C09088=1017.058,347.375,350.986,171.021,50.976,160.063
C09089=1017.051,347.128,351.023,171.013,50.980,160.063
C09090=1017.044,346.881,351.059,171.005,50.983,160.062
C09091=1017.036,346.634,351.096,170.997,50.986,160.061
C09092=1017.029,346.386,351.133,170.991,50.989,160.061
C09093=1017.022,346.139,351.168,170.983,50.992,160.060
C09094=1017.014,345.892,351.205,170.975,50.995,160.060
C09095=1017.007,345.644,351.241,170.967,50.998,160.059
C09096=1017.000,345.397,351.277,170.960,51.001,160.058
C09097=1016.992,345.150,351.314,170.953,51.004,160.058
C09098=1016.985,344.902,351.350,170.944,51.007,160.057
C09099=1016.978,344.655,351.386,170.938,51.010,160.057
C09100=1016.971,344.408,351.422,170.930,51.013,160.056
C09101=1016.964,344.161,351.458,170.922,51.017,160.056
C09102=1016.957,343.913,351.495,170.916,51.020,160.055
C09103=1016.949,343.666,351.531,170.908,51.023,160.054
C09104=1016.942,343.419,351.567,170.900,51.026,160.054
C09105=1016.935,343.171,351.604,170.892,51.029,160.053
C09106=1016.928,342.925,351.640,170.885,51.032,160.053
C09107=1016.921,342.677,351.675,170.878,51.036,160.052
C09108=1016.913,342.430,351.711,170.870,51.039,160.052
C09109=1016.907,342.182,351.748,170.863,51.042,160.051
C09110=1016.899,341.935,351.784,170.856,51.045,160.051
C09111=1016.892,341.687,351.819,170.848,51.049,160.050
C09112=1016.885,341.441,351.855,170.841,51.052,160.050
C09113=1016.878,341.193,351.892,170.833,51.055,160.049
C09114=1016.871,340.945,351.927,170.826,51.058,160.048
C09115=1016.864,340.699,351.963,170.819,51.061,160.048
C09116=1016.857,340.451,351.999,170.812,51.065,160.048
C09117=1016.850,340.204,352.034,170.804,51.069,160.047
C09118=1016.843,339.956,352.071,170.797,51.072,160.047
C09119=1016.836,339.709,352.106,170.790,51.075,160.046
C09120=1016.829,339.462,352.142,170.783,51.078,160.046
C09121=1016.822,339.214,352.178,170.775,51.081,160.045
C09122=1016.815,338.967,352.213,170.768,51.085,160.044
C09123=1016.808,338.720,352.249,170.761,51.088,160.044
C09124=1016.800,338.472,352.285,170.754,51.092,160.044
C09125=1016.793,338.225,352.320,170.746,51.096,160.043
C09126=1016.786,337.956,352.359,170.739,51.099,160.043
C09127=1016.778,337.686,352.397,170.731,51.103,160.042
C09128=1016.771,337.417,352.436,170.722,51.107,160.042
C09129=1016.763,337.148,352.474,170.715,51.111,160.041
C09130=1016.756,336.901,352.509,170.708,51.114,160.041
C09131=1016.749,336.653,352.545,170.701,51.117,160.040
C09132=1016.742,336.406,352.580,170.693,51.121,160.040
C09133=1016.735,336.158,352.615,170.687,51.125,160.040
C09134=1016.728,335.912,352.651,170.680,51.128,160.039
C09135=1016.721,335.664,352.686,170.672,51.132,160.039
C09136=1016.714,335.416,352.721,170.665,51.135,160.038
C09137=1016.707,335.169,352.757,170.658,51.139,160.038
C09138=1016.700,334.921,352.792,170.650,51.143,160.037
C09139=1016.694,334.674,352.827,170.644,51.146,160.037
C09140=1016.687,334.427,352.862,170.637,51.150,160.037
C09141=1016.680,334.179,352.897,170.630,51.153,160.036
C09142=1016.673,333.932,352.932,170.623,51.157,160.036
C09143=1016.667,333.685,352.967,170.616,51.161,160.035
C09144=1016.659,333.437,353.001,170.609,51.165,160.035
C09145=1016.652,333.189,353.037,170.601,51.168,160.035
C09146=1016.645,332.941,353.072,170.595,51.171,160.034
C09147=1016.639,332.694,353.107,170.588,51.176,160.034
C09148=1016.632,332.447,353.142,170.581,51.179,160.033
C09149=1016.625,332.199,353.177,170.574,51.183,160.033
C09150=1016.619,331.951,353.212,170.567,51.187,160.033
C09151=1016.611,331.704,353.246,170.560,51.190,160.032
C09152=1016.604,331.457,353.281,170.553,51.195,160.032
C09153=1016.598,331.209,353.316,170.547,51.198,160.032
C09154=1016.590,330.962,353.350,170.539,51.202,160.031
C09155=1016.584,330.714,353.385,170.532,51.206,160.031
C09156=1016.577,330.467,353.420,170.526,51.210,160.031
C09157=1016.570,330.220,353.453,170.518,51.214,160.031
C09158=1016.564,329.972,353.488,170.512,51.217,160.030
C09159=1016.557,329.724,353.523,170.505,51.221,160.030
C09160=1016.550,329.477,353.558,170.498,51.225,160.030
C09161=1016.543,329.229,353.592,170.491,51.229,160.029
C09162=1016.536,328.982,353.627,170.484,51.234,160.029
C09163=1016.530,328.734,353.661,170.477,51.237,160.029
C09164=1016.523,328.487,353.696,170.470,51.241,160.028
C09165=1016.517,328.240,353.730,170.464,51.245,160.028
C09166=1016.510,327.992,353.764,170.457,51.249,160.028
C09167=1016.503,327.744,353.799,170.451,51.253,160.028
C09168=1016.496,327.496,353.833,170.443,51.257,160.027
C09169=1016.490,327.248,353.868,170.437,51.261,160.027
C09170=1016.483,327.002,353.902,170.430,51.265,160.027
C09171=1016.476,326.754,353.936,170.423,51.269,160.026
C09172=1016.470,326.506,353.971,170.417,51.273,160.026
C09173=1016.463,326.258,354.005,170.409,51.277,160.026
C09174=1016.457,326.011,354.039,170.403,51.281,160.026
C09175=1016.450,325.764,354.072,170.396,51.285,160.025
C09176=1016.442,325.516,354.106,170.390,51.289,160.025
C09177=1016.437,325.269,354.140,170.383,51.293,160.025
C09178=1016.429,325.021,354.174,170.376,51.298,160.025
C09179=1016.422,324.773,354.208,170.370,51.302,160.024
C09180=1016.415,324.526,354.242,170.362,51.306,160.024
C09181=1016.408,324.279,354.275,170.357,51.311,160.024
C09182=1016.402,324.031,354.310,170.349,51.315,160.024
C09183=1016.395,323.783,354.343,170.342,51.319,160.024
C09184=1016.388,323.536,354.377,170.336,51.324,160.024
C09185=1016.381,323.288,354.410,170.329,51.328,160.023
C09186=1016.373,323.014,354.448,170.322,51.332,160.023
C09187=1016.367,322.741,354.485,170.314,51.337,160.023
C09188=1016.359,322.467,354.522,170.307,51.342,160.023
C09189=1016.352,322.194,354.559,170.300,51.346,160.022
C09190=1016.345,321.947,354.592,170.293,51.351,160.022
C09191=1016.339,321.699,354.627,170.286,51.355,160.022
C09192=1016.332,321.450,354.660,170.281,51.360,160.022
C09193=1016.325,321.203,354.693,170.273,51.364,160.022
C09194=1016.318,320.956,354.727,170.268,51.368,160.022
C09195=1016.312,320.708,354.760,170.260,51.373,160.021
C09196=1016.305,320.460,354.794,170.255,51.377,160.021
C09197=1016.298,320.213,354.828,170.247,51.381,160.021
C09198=1016.292,319.965,354.861,170.241,51.386,160.021
C09199=1016.285,319.718,354.894,170.235,51.391,160.021
C09200=1016.279,319.470,354.928,170.228,51.395,160.020
C09201=1016.272,319.222,354.961,170.222,51.399,160.020
C09202=1016.266,318.975,354.994,170.215,51.404,160.020
C09203=1016.259,318.727,355.028,170.209,51.408,160.020
C09204=1016.252,318.479,355.061,170.202,51.413,160.020
C09205=1016.246,318.231,355.094,170.196,51.417,160.020
C09206=1016.240,317.984,355.128,170.189,51.422,160.020
C09207=1016.233,317.736,355.161,170.183,51.426,160.020
C09208=1016.226,317.489,355.194,170.176,51.431,160.020
C09209=1016.221,317.241,355.228,170.170,51.435,160.019
C09210=1016.214,316.993,355.261,170.163,51.440,160.019
C09211=1016.207,316.745,355.294,170.157,51.445,160.019
C09212=1016.201,316.498,355.327,170.151,51.449,160.019
C09213=1016.195,316.250,355.360,170.144,51.453,160.019
C09214=1016.189,316.003,355.394,170.138,51.458,160.019
C09215=1016.182,315.755,355.427,170.131,51.463,160.019
C09216=1016.176,315.507,355.460,170.125,51.467,160.019
C09217=1016.169,315.259,355.492,170.119,51.472,160.019
C09218=1016.163,315.012,355.525,170.113,51.477,160.019
C09219=1016.156,314.764,355.560,170.106,51.481,160.018
C09220=1016.150,314.516,355.592,170.100,51.486,160.018
C09221=1016.144,314.269,355.625,170.093,51.491,160.018
C09222=1016.138,314.021,355.658,170.087,51.495,160.018
C09223=1016.131,313.774,355.691,170.080,51.500,160.018
C09224=1016.125,313.525,355.724,170.075,51.504,160.018
C09225=1016.119,313.277,355.757,170.068,51.509,160.018
C09226=1016.113,313.030,355.790,170.062,51.513,160.018
C09227=1016.106,312.783,355.823,170.055,51.518,160.018
C09228=1016.100,312.535,355.856,170.050,51.523,160.018
C09229=1016.094,312.287,355.889,170.043,51.528,160.018
C09230=1016.088,312.040,355.922,170.037,51.533,160.018
C09231=1016.082,311.792,355.955,170.031,51.538,160.018
C09232=1016.075,311.544,355.988,170.025,51.542,160.018
C09233=1016.069,311.297,356.020,170.018,51.547,160.018
C09234=1016.064,311.048,356.053,170.012,51.552,160.018
C09235=1016.057,310.801,356.086,170.005,51.557,160.017
C09236=1016.051,310.553,356.118,170.000,51.561,160.017
C09237=1016.045,310.306,356.151,169.993,51.566,160.017
C09238=1016.039,310.058,356.184,169.988,51.571,160.018
C09239=1016.032,309.810,356.217,169.981,51.576,160.017
C09240=1016.027,309.563,356.250,169.975,51.581,160.017
C09241=1016.021,309.314,356.282,169.968,51.585,160.017
C09242=1016.014,309.067,356.314,169.963,51.591,160.017
C09243=1016.008,308.819,356.346,169.956,51.595,160.017
C09244=1016.001,308.572,356.378,169.951,51.601,160.018
C09245=1015.995,308.323,356.410,169.944,51.606,160.017
C09246=1015.987,308.055,356.445,169.938,51.611,160.018
C09247=1015.980,307.787,356.480,169.931,51.617,160.018
C09248=1015.973,307.520,356.515,169.924,51.623,160.018
C09249=1015.966,307.252,356.550,169.917,51.628,160.018
C09250=1015.960,307.003,356.582,169.912,51.633,160.018
C09251=1015.953,306.756,356.613,169.905,51.638,160.018
C09252=1015.947,306.508,356.646,169.899,51.644,160.018
C09253=1015.940,306.260,356.677,169.893,51.648,160.018
C09254=1015.934,306.012,356.709,169.887,51.654,160.018
C09255=1015.928,305.765,356.740,169.882,51.659,160.018
C09256=1015.922,305.517,356.773,169.875,51.664,160.018
C09257=1015.915,305.269,356.805,169.868,51.669,160.018
C09258=1015.909,305.021,356.837,169.863,51.675,160.018
C09259=1015.903,304.773,356.869,169.856,51.680,160.018
C09260=1015.896,304.525,356.901,169.851,51.685,160.018
C09261=1015.890,304.277,356.933,169.845,51.690,160.019
C09262=1015.884,304.030,356.964,169.838,51.696,160.019
C09263=1015.878,303.782,356.996,169.832,51.700,160.019
C09264=1015.871,303.534,357.027,169.826,51.706,160.019
C09265=1015.865,303.286,357.059,169.821,51.711,160.019
C09266=1015.859,303.038,357.091,169.814,51.717,160.019
C09267=1015.853,302.790,357.122,169.808,51.722,160.019
C09268=1015.846,302.543,357.155,169.803,51.727,160.019
C09269=1015.840,302.295,357.187,169.796,51.733,160.019
C09270=1015.834,302.047,357.219,169.790,51.738,160.019
C09271=1015.828,301.799,357.250,169.784,51.743,160.019
C09272=1015.822,301.551,357.282,169.779,51.748,160.020
C09273=1015.815,301.303,357.313,169.772,51.754,160.020
C09274=1015.809,301.055,357.345,169.766,51.759,160.020
C09275=1015.803,300.808,357.376,169.761,51.765,160.020
C09276=1015.798,300.559,357.408,169.754,51.770,160.020
C09277=1015.791,300.311,357.439,169.749,51.775,160.020
C09278=1015.785,300.064,357.471,169.743,51.781,160.020
C09279=1015.779,299.816,357.502,169.737,51.786,160.021
C09280=1015.773,299.568,357.534,169.731,51.792,160.021
C09281=1015.767,299.320,357.565,169.725,51.797,160.021
C09282=1015.761,299.072,357.597,169.719,51.803,160.021
C09283=1015.755,298.825,357.629,169.713,51.808,160.021
C09284=1015.749,298.576,357.660,169.708,51.813,160.021
C09285=1015.743,298.328,357.691,169.702,51.820,160.022
C09286=1015.737,298.081,357.723,169.696,51.825,160.022
C09287=1015.731,297.832,357.755,169.690,51.830,160.022
C09288=1015.725,297.585,357.785,169.684,51.836,160.022
C09289=1015.719,297.336,357.817,169.678,51.841,160.022
C09290=1015.713,297.089,357.848,169.672,51.847,160.022
C09291=1015.707,296.841,357.880,169.667,51.853,160.023
C09292=1015.701,296.593,357.910,169.661,51.858,160.023
C09293=1015.695,296.345,357.943,169.655,51.864,160.023
C09294=1015.689,296.098,357.974,169.649,51.869,160.023
C09295=1015.683,295.849,358.005,169.643,51.875,160.023
C09296=1015.677,295.602,358.036,169.638,51.881,160.023
C09297=1015.671,295.353,358.067,169.631,51.886,160.024
C09298=1015.665,295.106,358.098,169.626,51.891,160.024
C09299=1015.659,294.857,358.130,169.620,51.898,160.024
C09300=1015.654,294.609,358.161,169.615,51.903,160.024
C09301=1015.648,294.362,358.192,169.608,51.908,160.024
C09302=1015.642,294.113,358.224,169.602,51.915,160.025
C09303=1015.636,293.866,358.255,169.597,51.920,160.025
C09304=1015.631,293.617,358.286,169.591,51.926,160.025
C09305=1015.624,293.370,358.317,169.586,51.931,160.025
C09306=1015.619,293.120,358.348,169.579,51.937,160.025
C09307=1015.613,292.869,358.380,169.575,51.943,160.026
C09308=1015.607,292.619,358.411,169.568,51.949,160.026
C09309=1015.601,292.370,358.442,169.562,51.955,160.026
C09310=1015.595,292.122,358.473,169.557,51.960,160.026
C09311=1015.589,291.873,358.503,169.551,51.966,160.027
C09312=1015.583,291.625,358.534,169.545,51.973,160.027
C09313=1015.578,291.378,358.565,169.540,51.978,160.027
C09314=1015.571,291.129,358.596,169.534,51.984,160.027
C09315=1015.565,290.882,358.626,169.528,51.990,160.028
C09316=1015.560,290.634,358.657,169.523,51.996,160.028
C09317=1015.553,290.385,358.688,169.517,52.002,160.028
C09318=1015.547,290.137,358.718,169.511,52.008,160.029
C09319=1015.541,289.890,358.748,169.505,52.013,160.029
C09320=1015.535,289.641,358.779,169.500,52.020,160.029
C09321=1015.529,289.393,358.809,169.494,52.026,160.029
C09322=1015.523,289.145,358.840,169.489,52.032,160.030
C09323=1015.517,288.897,358.870,169.483,52.038,160.030
C09324=1015.511,288.649,358.901,169.477,52.044,160.030
C09325=1015.505,288.401,358.931,169.472,52.050,160.030
C09326=1015.500,288.153,358.962,169.466,52.056,160.031
C09327=1015.494,287.905,358.993,169.460,52.062,160.031
C09328=1015.488,287.657,359.023,169.455,52.068,160.031
C09329=1015.482,287.409,359.053,169.449,52.074,160.032
C09330=1015.476,287.161,359.084,169.443,52.081,160.032
C09331=1015.471,286.913,359.113,169.438,52.087,160.032
C09332=1015.465,286.664,359.144,169.432,52.093,160.033
C09333=1015.459,286.416,359.174,169.426,52.099,160.033
C09334=1015.453,286.168,359.205,169.421,52.105,160.033
C09335=1015.446,285.921,359.235,169.416,52.112,160.034
C09336=1015.441,285.673,359.264,169.410,52.118,160.034
C09337=1015.435,285.425,359.295,169.404,52.124,160.034
C09338=1015.429,285.176,359.325,169.399,52.130,160.035
C09339=1015.423,284.928,359.355,169.393,52.136,160.035
C09340=1015.417,284.680,359.385,169.387,52.143,160.035
C09341=1015.411,284.432,359.416,169.382,52.149,160.036
C09342=1015.406,284.184,359.445,169.376,52.155,160.036
C09343=1015.400,283.936,359.476,169.371,52.162,160.037
C09344=1015.394,283.688,359.505,169.365,52.168,160.037
C09345=1015.388,283.440,359.535,169.360,52.174,160.037
C09346=1015.382,283.192,359.565,169.354,52.180,160.038
C09347=1015.377,282.944,359.595,169.349,52.187,160.038
C09348=1015.370,282.696,359.625,169.343,52.194,160.038
C09349=1015.364,282.447,359.655,169.338,52.200,160.039
C09350=1015.359,282.199,359.684,169.332,52.206,160.039
C09351=1015.353,281.951,359.715,169.327,52.213,160.040
C09352=1015.346,281.703,359.744,169.321,52.219,160.040
C09353=1015.341,281.455,359.774,169.316,52.225,160.040
C09354=1015.335,281.206,359.804,169.310,52.232,160.041
C09355=1015.329,280.958,359.833,169.304,52.238,160.041
C09356=1015.323,280.710,359.863,169.299,52.245,160.042
C09357=1015.318,280.462,359.893,169.294,52.251,160.042
C09358=1015.312,280.213,359.922,169.288,52.258,160.042
C09359=1015.305,279.966,359.952,169.283,52.265,160.043
C09360=1015.300,279.718,359.982,169.277,52.271,160.043
C09361=1015.294,279.469,360.011,169.271,52.278,160.044
C09362=1015.289,279.226,360.041,169.266,52.284,160.044
C09363=1015.283,278.984,360.069,169.261,52.290,160.044
C09364=1015.278,278.741,360.098,169.256,52.297,160.045
C09365=1015.272,278.498,360.127,169.250,52.303,160.045
C09366=1015.267,278.255,360.156,169.245,52.310,160.046
C09367=1015.261,278.012,360.185,169.240,52.316,160.046
C09368=1015.255,277.769,360.214,169.234,52.323,160.046
C09369=1015.249,277.526,360.243,169.230,52.329,160.047
C09370=1015.244,277.278,360.273,169.224,52.336,160.047
C09371=1015.239,277.030,360.302,169.218,52.343,160.048
C09372=1015.232,276.782,360.332,169.213,52.350,160.048
C09373=1015.227,276.534,360.361,169.208,52.355,160.049
C09374=1015.221,276.285,360.391,169.203,52.363,160.049
C09375=1015.215,276.037,360.420,169.197,52.370,160.050
C09376=1015.210,275.789,360.449,169.191,52.376,160.050
C09377=1015.204,275.541,360.478,169.186,52.383,160.050
C09378=1015.199,275.293,360.508,169.180,52.390,160.051
C09379=1015.192,275.045,360.537,169.176,52.397,160.052
C09380=1015.187,274.796,360.566,169.170,52.403,160.052
C09381=1015.181,274.548,360.595,169.165,52.410,160.052
C09382=1015.176,274.300,360.625,169.159,52.417,160.053
C09383=1015.170,274.052,360.653,169.154,52.424,160.053
C09384=1015.164,273.803,360.683,169.148,52.431,160.054
C09385=1015.158,273.555,360.712,169.143,52.438,160.054
C09386=1015.152,273.307,360.741,169.138,52.445,160.055
C09387=1015.147,273.059,360.770,169.133,52.451,160.055
C09388=1015.141,272.810,360.798,169.127,52.458,160.056
C09389=1015.135,272.562,360.828,169.122,52.465,160.056
C09390=1015.129,272.314,360.857,169.116,52.472,160.057
C09391=1015.124,272.066,360.886,169.111,52.479,160.057
C09392=1015.118,271.817,360.915,169.105,52.486,160.058
C09393=1015.113,271.569,360.944,169.101,52.493,160.059
C09394=1015.107,271.321,360.973,169.096,52.500,160.059
C09395=1015.101,271.073,361.001,169.090,52.507,160.060
C09396=1015.096,270.824,361.031,169.085,52.514,160.060
C09397=1015.090,270.577,361.060,169.079,52.521,160.061
C09398=1015.084,270.328,361.088,169.074,52.528,160.061
C09399=1015.078,270.080,361.118,169.068,52.535,160.062
C09400=1015.073,269.832,361.146,169.063,52.543,160.062
C09401=1015.068,269.583,361.175,169.058,52.550,160.063
C09402=1015.061,269.335,361.204,169.054,52.556,160.063
C09403=1015.056,269.087,361.232,169.048,52.564,160.064
C09404=1015.051,268.838,361.262,169.043,52.571,160.064
C09405=1015.045,268.590,361.290,169.037,52.578,160.065
C09406=1015.039,268.342,361.319,169.032,52.585,160.066
C09407=1015.033,268.094,361.347,169.027,52.592,160.066
C09408=1015.028,267.845,361.375,169.021,52.599,160.067
C09409=1015.022,267.597,361.405,169.016,52.607,160.067
C09410=1015.016,267.348,361.433,169.011,52.614,160.068
C09411=1015.011,267.100,361.461,169.006,52.621,160.068
C09412=1015.005,266.852,361.490,169.000,52.628,160.069
C09413=1015.000,266.604,361.519,168.995,52.636,160.070
C09414=1014.994,266.355,361.547,168.990,52.643,160.070
C09415=1014.988,266.108,361.576,168.984,52.650,160.071
C09416=1014.982,265.859,361.604,168.980,52.658,160.071
C09417=1014.977,265.611,361.632,168.974,52.665,160.072
C09418=1014.971,265.363,361.661,168.969,52.673,160.073
C09419=1014.966,265.114,361.689,168.964,52.680,160.073
C09420=1014.960,264.866,361.718,168.958,52.687,160.074
C09421=1014.955,264.617,361.746,168.953,52.695,160.074
C09422=1014.949,264.376,361.773,168.949,52.701,160.075
C09423=1014.943,264.136,361.801,168.944,52.709,160.076
C09424=1014.939,263.895,361.828,168.939,52.716,160.076
C09425=1014.933,263.654,361.855,168.933,52.723,160.077
C09426=1014.928,263.414,361.882,168.928,52.731,160.077
C09427=1014.922,263.174,361.910,168.924,52.738,160.078
C09428=1014.916,262.933,361.937,168.918,52.745,160.078
C09429=1014.911,262.692,361.965,168.914,52.753,160.079
C09430=1014.905,262.443,361.993,168.908,52.760,160.080
C09431=1014.900,262.195,362.021,168.903,52.767,160.080
C09432=1014.895,261.947,362.049,168.898,52.775,160.081
C09433=1014.889,261.698,362.077,168.893,52.782,160.082
C09434=1014.883,261.450,362.105,168.888,52.790,160.082
C09435=1014.877,261.202,362.134,168.883,52.798,160.083
C09436=1014.872,260.954,362.162,168.878,52.805,160.084
C09437=1014.867,260.705,362.190,168.873,52.813,160.084
C09438=1014.861,260.457,362.218,168.868,52.820,160.085
C09439=1014.855,260.209,362.246,168.863,52.828,160.086
C09440=1014.850,259.960,362.274,168.857,52.835,160.086
C09441=1014.844,259.711,362.301,168.852,52.843,160.087
C09442=1014.839,259.463,362.329,168.846,52.851,160.088
C09443=1014.834,259.215,362.357,168.841,52.859,160.088
C09444=1014.827,258.967,362.385,168.837,52.867,160.089
C09445=1014.822,258.719,362.413,168.832,52.875,160.090
C09446=1014.816,258.470,362.440,168.827,52.882,160.091
C09447=1014.810,258.222,362.468,168.822,52.890,160.091
C09448=1014.805,257.973,362.495,168.816,52.898,160.092
C09449=1014.799,257.725,362.523,168.811,52.906,160.093
C09450=1014.793,257.476,362.551,168.806,52.914,160.093
C09451=1014.787,257.228,362.578,168.801,52.922,160.094
C09452=1014.782,256.980,362.606,168.796,52.929,160.095
C09453=1014.776,256.731,362.633,168.790,52.938,160.095
C09454=1014.770,256.483,362.661,168.785,52.945,160.096
C09455=1014.765,256.234,362.688,168.780,52.953,160.097
C09456=1014.759,255.986,362.715,168.775,52.961,160.098
C09457=1014.753,255.737,362.743,168.770,52.969,160.098
C09458=1014.748,255.489,362.771,168.765,52.978,160.099
C09459=1014.742,255.241,362.797,168.760,52.985,160.100
C09460=1014.737,254.993,362.825,168.755,52.993,160.101
C09461=1014.731,254.743,362.853,168.750,53.001,160.101
C09462=1014.726,254.495,362.880,168.744,53.009,160.102
C09463=1014.720,254.247,362.908,168.740,53.018,160.103
C09464=1014.714,253.998,362.934,168.735,53.026,160.104
C09465=1014.709,253.750,362.962,168.730,53.033,160.104
C09466=1014.703,253.501,362.990,168.725,53.041,160.105
C09467=1014.698,253.253,363.016,168.719,53.049,160.106
C09468=1014.692,253.005,363.044,168.715,53.058,160.107
C09469=1014.687,252.756,363.071,168.710,53.066,160.107
C09470=1014.682,252.508,363.098,168.705,53.074,160.108
C09471=1014.676,252.260,363.126,168.700,53.082,160.109
C09472=1014.670,252.011,363.153,168.695,53.090,160.110
C09473=1014.665,251.762,363.181,168.690,53.098,160.110
C09474=1014.659,251.513,363.207,168.685,53.107,160.111
C09475=1014.654,251.265,363.235,168.679,53.115,160.112
C09476=1014.649,251.017,363.262,168.674,53.123,160.113
C09477=1014.643,250.768,363.289,168.670,53.131,160.114
C09478=1014.638,250.520,363.316,168.664,53.139,160.114
C09479=1014.632,250.272,363.344,168.660,53.148,160.115
C09480=1014.627,250.023,363.371,168.655,53.156,160.116
C09481=1014.622,249.775,363.398,168.650,53.164,160.117
C09482=1014.616,249.533,363.425,168.645,53.172,160.118
C09483=1014.611,249.291,363.451,168.641,53.180,160.118
C09484=1014.605,249.050,363.478,168.636,53.188,160.119
C09485=1014.600,248.808,363.504,168.630,53.196,160.120
C09486=1014.595,248.566,363.529,168.625,53.204,160.121
C09487=1014.590,248.325,363.556,168.620,53.212,160.121
C09488=1014.584,248.083,363.582,168.616,53.220,160.122
C09489=1014.579,247.841,363.609,168.611,53.229,160.123
C09490=1014.574,247.593,363.636,168.606,53.237,160.124
C09491=1014.568,247.344,363.663,168.602,53.245,160.125
C09492=1014.563,247.096,363.690,168.596,53.253,160.125
C09493=1014.558,246.847,363.717,168.592,53.262,160.126
C09494=1014.552,246.599,363.744,168.587,53.270,160.127
C09495=1014.547,246.350,363.771,168.581,53.279,160.128
C09496=1014.542,246.102,363.797,168.577,53.287,160.129
C09497=1014.537,245.854,363.825,168.572,53.295,160.129
C09498=1014.532,245.605,363.852,168.567,53.304,160.130
C09499=1014.526,245.357,363.879,168.562,53.312,160.131
C09500=1014.521,245.108,363.906,168.557,53.320,160.132
C09501=1014.515,244.860,363.932,168.552,53.329,160.133
C09502=1014.510,244.611,363.960,168.547,53.338,160.134
C09503=1014.505,244.362,363.987,168.543,53.346,160.134
C09504=1014.499,244.114,364.014,168.537,53.355,160.135
C09505=1014.494,243.865,364.041,168.533,53.363,160.136
C09506=1014.489,243.618,364.067,168.528,53.371,160.137
C09507=1014.484,243.368,364.094,168.522,53.380,160.138
C09508=1014.479,243.120,364.120,168.518,53.389,160.139
C09509=1014.474,242.871,364.148,168.514,53.397,160.140
C09510=1014.469,242.623,364.175,168.508,53.406,160.141
C09511=1014.463,242.374,364.201,168.503,53.414,160.141
C09512=1014.458,242.127,364.228,168.498,53.423,160.142
C09513=1014.452,241.878,364.254,168.494,53.432,160.143
C09514=1014.447,241.629,364.281,168.488,53.440,160.144
C09515=1014.441,241.381,364.308,168.484,53.449,160.145
C09516=1014.436,241.132,364.333,168.480,53.458,160.146
C09517=1014.431,240.884,364.360,168.474,53.467,160.147
C09518=1014.426,240.635,364.386,168.470,53.475,160.148
C09519=1014.420,240.386,364.413,168.464,53.484,160.148
C09520=1014.414,240.138,364.440,168.460,53.493,160.149
C09521=1014.410,239.889,364.466,168.455,53.502,160.150
C09522=1014.404,239.641,364.492,168.450,53.510,160.151
C09523=1014.399,239.392,364.518,168.445,53.519,160.152
C09524=1014.394,239.143,364.546,168.440,53.528,160.153
C09525=1014.388,238.894,364.572,168.436,53.538,160.154
C09526=1014.383,238.647,364.598,168.431,53.546,160.155
C09527=1014.378,238.398,364.624,168.426,53.555,160.156
C09528=1014.372,238.149,364.650,168.421,53.564,160.157
C09529=1014.367,237.901,364.676,168.416,53.573,160.158
C09530=1014.361,237.653,364.703,168.411,53.582,160.159
C09531=1014.356,237.404,364.729,168.407,53.591,160.160
C09532=1014.351,237.156,364.754,168.401,53.600,160.160
C09533=1014.345,236.907,364.781,168.397,53.609,160.161
C09534=1014.340,236.658,364.807,168.392,53.618,160.162
C09535=1014.334,236.409,364.833,168.387,53.627,160.163
C09536=1014.330,236.161,364.858,168.382,53.636,160.164
C09537=1014.324,235.913,364.885,168.378,53.646,160.165
C09538=1014.318,235.664,364.911,168.373,53.654,160.166
C09539=1014.313,235.415,364.936,168.368,53.663,160.167
C09540=1014.308,235.166,364.962,168.363,53.673,160.168
C09541=1014.302,234.918,364.989,168.359,53.681,160.169
C09542=1014.297,234.673,365.015,168.353,53.690,160.170
C09543=1014.293,234.428,365.040,168.349,53.700,160.171
C09544=1014.287,234.183,365.065,168.344,53.709,160.172
C09545=1014.282,233.938,365.091,168.340,53.717,160.173
C09546=1014.277,233.693,365.116,168.335,53.727,160.174
C09547=1014.271,233.448,365.141,168.329,53.736,160.175
C09548=1014.266,233.202,365.167,168.326,53.745,160.176
C09549=1014.261,232.957,365.193,168.320,53.754,160.177
C09550=1014.256,232.708,365.219,168.316,53.763,160.178
C09551=1014.251,232.460,365.244,168.311,53.773,160.179
C09552=1014.245,232.211,365.270,168.306,53.783,160.180
C09553=1014.240,231.963,365.295,168.302,53.791,160.181
C09554=1014.234,231.715,365.322,168.297,53.801,160.182
C09555=1014.229,231.466,365.347,168.292,53.810,160.183
C09556=1014.224,231.217,365.373,168.288,53.819,160.184
C09557=1014.219,230.969,365.399,168.283,53.828,160.185
C09558=1014.213,230.720,365.425,168.278,53.838,160.186
C09559=1014.208,230.472,365.450,168.273,53.848,160.187
C09560=1014.203,230.223,365.476,168.269,53.856,160.188
C09561=1014.198,229.974,365.501,168.264,53.866,160.189
C09562=1014.193,229.725,365.527,168.259,53.876,160.190
C09563=1014.188,229.477,365.553,168.255,53.885,160.191
C09564=1014.183,229.228,365.579,168.250,53.894,160.192
C09565=1014.177,228.980,365.603,168.245,53.904,160.193
C09566=1014.171,228.731,365.629,168.240,53.914,160.194
C09567=1014.167,228.482,365.655,168.235,53.923,160.195
C09568=1014.161,228.233,365.681,168.231,53.932,160.196
C09569=1014.157,227.984,365.706,168.226,53.942,160.197
C09570=1014.150,227.736,365.731,168.221,53.952,160.198
C09571=1014.146,227.488,365.757,168.216,53.961,160.199
C09572=1014.140,227.239,365.783,168.211,53.970,160.200
C09573=1014.135,226.990,365.807,168.207,53.980,160.202
C09574=1014.130,226.742,365.832,168.202,53.990,160.203
C09575=1014.124,226.493,365.858,168.198,53.999,160.204
C09576=1014.120,226.244,365.884,168.193,54.009,160.205
C09577=1014.114,225.995,365.909,168.188,54.019,160.206
C09578=1014.109,225.747,365.934,168.183,54.029,160.207
C09579=1014.104,225.499,365.960,168.178,54.038,160.208
C09580=1014.098,225.249,365.984,168.174,54.048,160.209
C09581=1014.093,225.001,366.010,168.170,54.058,160.210
C09582=1014.087,224.752,366.035,168.165,54.067,160.211
C09583=1014.082,224.503,366.060,168.160,54.077,160.212
C09584=1014.077,224.255,366.084,168.155,54.087,160.213
C09585=1014.072,224.006,366.110,168.151,54.097,160.215
C09586=1014.067,223.757,366.135,168.146,54.106,160.216
C09587=1014.061,223.509,366.160,168.141,54.117,160.217
C09588=1014.056,223.259,366.185,168.137,54.127,160.218
C09589=1014.051,223.011,366.210,168.132,54.137,160.219
C09590=1014.046,222.763,366.235,168.127,54.146,160.220
C09591=1014.040,222.513,366.260,168.122,54.156,160.221
C09592=1014.035,222.265,366.285,168.118,54.166,160.222
C09593=1014.030,222.016,366.310,168.113,54.176,160.223
C09594=1014.025,221.767,366.335,168.108,54.186,160.225
C09595=1014.019,221.519,366.360,168.104,54.196,160.226
C09596=1014.014,221.271,366.385,168.099,54.206,160.227
C09597=1014.009,221.021,366.410,168.094,54.216,160.228
C09598=1014.004,220.772,366.435,168.090,54.226,160.229
C09599=1013.998,220.524,366.460,168.085,54.236,160.230
C09600=1013.994,220.275,366.485,168.080,54.246,160.231
C09601=1013.988,220.026,366.509,168.076,54.256,160.232
C09602=1013.983,219.778,366.535,168.071,54.266,160.234
C09603=1013.978,219.529,366.559,168.067,54.276,160.235
C09604=1013.973,219.280,366.584,168.062,54.286,160.236
C09605=1013.969,219.032,366.609,168.057,54.296,160.237
C09606=1013.962,218.782,366.634,168.053,54.306,160.238
C09607=1013.957,218.532,366.659,168.048,54.316,160.239
C09608=1013.952,218.282,366.683,168.044,54.326,160.241
C09609=1013.947,218.032,366.709,168.039,54.336,160.242
C09610=1013.942,217.783,366.734,168.035,54.347,160.243
C09611=1013.937,217.535,366.758,168.030,54.357,160.244
C09612=1013.931,217.287,366.783,168.025,54.368,160.245
C09613=1013.926,217.038,366.807,168.020,54.377,160.246
C09614=1013.922,216.789,366.832,168.016,54.388,160.248
C09615=1013.916,216.540,366.856,168.011,54.398,160.249
C09616=1013.910,216.291,366.881,168.007,54.408,160.250
C09617=1013.905,216.043,366.905,168.002,54.418,160.251
C09618=1013.901,215.794,366.930,167.997,54.429,160.252
C09619=1013.895,215.545,366.954,167.992,54.440,160.254
C09620=1013.890,215.297,366.978,167.988,54.449,160.255
C09621=1013.885,215.048,367.003,167.984,54.460,160.256
C09622=1013.879,214.799,367.027,167.979,54.470,160.257
C09623=1013.874,214.550,367.052,167.975,54.480,160.259
C09624=1013.869,214.301,367.076,167.969,54.491,160.260
C09625=1013.864,214.053,367.101,167.965,54.501,160.261
C09626=1013.859,213.803,367.124,167.960,54.512,160.262
C09627=1013.854,213.555,367.149,167.956,54.522,160.263
C09628=1013.849,213.306,367.173,167.951,54.533,160.265
C09629=1013.843,213.057,367.198,167.946,54.543,160.266
C09630=1013.838,212.809,367.222,167.942,54.554,160.267
C09631=1013.833,212.560,367.246,167.938,54.564,160.268
C09632=1013.828,212.311,367.271,167.933,54.574,160.269
C09633=1013.823,212.063,367.295,167.928,54.585,160.271
C09634=1013.818,211.813,367.319,167.924,54.596,160.272
C09635=1013.813,211.565,367.343,167.920,54.606,160.273
C09636=1013.808,211.316,367.368,167.914,54.617,160.274
C09637=1013.803,211.067,367.392,167.910,54.627,160.276
C09638=1013.798,210.819,367.416,167.905,54.638,160.277
C09639=1013.792,210.570,367.441,167.901,54.648,160.278
C09640=1013.787,210.321,367.464,167.896,54.659,160.279
C09641=1013.783,210.072,367.489,167.892,54.670,160.281
C09642=1013.777,209.824,367.513,167.888,54.681,160.282
C09643=1013.772,209.575,367.537,167.883,54.691,160.283
C09644=1013.767,209.326,367.561,167.878,54.702,160.284
C09645=1013.762,209.077,367.585,167.874,54.712,160.286
C09646=1013.757,208.829,367.610,167.870,54.723,160.287
C09647=1013.752,208.579,367.633,167.864,54.734,160.288
C09648=1013.746,208.331,367.657,167.860,54.744,160.290
C09649=1013.741,208.082,367.681,167.855,54.755,160.291
C09650=1013.736,207.833,367.705,167.851,54.766,160.292
C09651=1013.731,207.584,367.729,167.847,54.777,160.293
C09652=1013.726,207.335,367.753,167.842,54.788,160.295
C09653=1013.720,207.087,367.777,167.837,54.798,160.296
C09654=1013.716,206.838,367.800,167.832,54.809,160.297
C09655=1013.711,206.590,367.825,167.829,54.821,160.299
C09656=1013.706,206.340,367.848,167.824,54.831,160.300
C09657=1013.700,206.092,367.872,167.819,54.842,160.301
C09658=1013.695,205.843,367.896,167.815,54.853,160.303
C09659=1013.690,205.594,367.920,167.810,54.864,160.304
C09660=1013.685,205.345,367.944,167.806,54.875,160.305
C09661=1013.681,205.096,367.967,167.801,54.886,160.306
C09662=1013.675,204.855,367.990,167.797,54.896,160.308
C09663=1013.670,204.612,368.014,167.792,54.907,160.309
C09664=1013.665,204.370,368.037,167.788,54.918,160.310
C09665=1013.661,204.128,368.060,167.783,54.929,160.312
C09666=1013.655,203.886,368.082,167.779,54.939,160.313
C09667=1013.650,203.644,368.105,167.775,54.950,160.314
C09668=1013.646,203.402,368.128,167.770,54.961,160.315
C09669=1013.640,203.160,368.151,167.766,54.972,160.317
C09670=1013.623,202.089,368.245,167.234,54.871,160.172
C09671=1013.619,201.841,368.267,167.229,54.883,160.173
C09672=1013.614,201.592,368.289,167.224,54.896,160.174
C09673=1013.611,201.342,368.311,167.219,54.908,160.176
C09674=1013.607,201.094,368.333,167.214,54.920,160.177
C09675=1013.603,200.844,368.354,167.210,54.932,160.179
C09676=1013.599,200.596,368.376,167.205,54.944,160.180
C09677=1013.595,200.347,368.399,167.201,54.956,160.182
C09678=1013.590,200.097,368.420,167.195,54.969,160.183
C09679=1013.587,199.849,368.442,167.191,54.980,160.184
C09680=1013.583,199.599,368.464,167.186,54.993,160.186
C09681=1013.579,199.351,368.485,167.182,55.005,160.187
C09682=1013.575,199.101,368.507,167.177,55.017,160.189
C09683=1013.571,198.852,368.529,167.173,55.029,160.190
C09684=1013.567,198.603,368.550,167.168,55.041,160.192
C09685=1013.562,198.355,368.572,167.162,55.053,160.193
C09686=1013.559,198.105,368.594,167.158,55.066,160.194
C09687=1013.555,197.856,368.614,167.153,55.078,160.196
C09688=1013.550,197.607,368.636,167.149,55.090,160.197
C09689=1013.546,197.359,368.657,167.144,55.102,160.199
C09690=1013.542,197.109,368.679,167.139,55.115,160.200
C09691=1013.538,196.860,368.700,167.135,55.127,160.201
C09692=1013.534,196.611,368.721,167.130,55.139,160.203
C09693=1013.530,196.363,368.742,167.126,55.151,160.204
C09694=1013.526,196.113,368.764,167.122,55.164,160.206
C09695=1013.521,195.863,368.785,167.117,55.176,160.207
C09696=1013.517,195.615,368.806,167.113,55.188,160.209
C09697=1013.514,195.365,368.828,167.107,55.200,160.210
C09698=1013.509,195.117,368.849,167.103,55.213,160.212
C09699=1013.505,194.867,368.870,167.098,55.225,160.213
C09700=1013.501,194.619,368.891,167.093,55.237,160.214
C09701=1013.497,194.369,368.913,167.089,55.249,160.216
C09702=1013.493,194.120,368.934,167.085,55.261,160.217
C09703=1013.489,193.871,368.954,167.081,55.274,160.219
C09704=1013.484,193.623,368.976,167.076,55.286,160.220
C09705=1013.481,193.374,368.998,167.072,55.298,160.222
C09706=1013.477,193.124,369.019,167.067,55.310,160.223
C09707=1013.473,192.875,369.040,167.062,55.322,160.225
C09708=1013.469,192.626,369.061,167.058,55.335,160.226
C09709=1013.465,192.377,369.082,167.054,55.347,160.228
C09710=1013.461,192.128,369.103,167.050,55.359,160.229
C09711=1013.457,191.879,369.124,167.045,55.371,160.231
C09712=1013.454,191.630,369.145,167.040,55.383,160.232
C09713=1013.449,191.380,369.167,167.036,55.396,160.234
C09714=1013.445,191.132,369.187,167.032,55.407,160.235
C09715=1013.441,190.882,369.208,167.027,55.419,160.236
C09716=1013.437,190.633,369.230,167.023,55.432,160.238
C09717=1013.433,190.384,369.251,167.018,55.444,160.239
C09718=1013.429,190.135,369.272,167.014,55.456,160.241
C09719=1013.426,189.886,369.293,167.010,55.468,160.242
C09720=1013.422,189.637,369.314,167.005,55.480,160.244
C09721=1013.417,189.388,369.335,167.001,55.493,160.245
C09722=1013.413,189.139,369.356,166.996,55.505,160.247
C09723=1013.410,188.890,369.377,166.992,55.517,160.248
C09724=1013.406,188.641,369.398,166.988,55.529,160.250
C09725=1013.402,188.392,369.419,166.983,55.541,160.251
C09726=1013.398,188.143,369.440,166.979,55.553,160.252
C09727=1013.394,187.893,369.462,166.975,55.566,160.254
C09728=1013.390,187.645,369.482,166.970,55.578,160.255
C09729=1013.386,187.396,369.503,166.966,55.590,160.257
C09730=1013.382,187.146,369.524,166.962,55.601,160.258
C09731=1013.378,186.868,369.548,166.957,55.615,160.260
C09732=1013.374,186.589,369.571,166.953,55.629,160.262
C09733=1013.369,186.309,369.595,166.948,55.642,160.263
C09734=1013.365,186.030,369.618,166.943,55.656,160.265
C09735=1013.361,185.781,369.638,166.939,55.668,160.266
C09736=1013.357,185.532,369.659,166.935,55.681,160.268
C09737=1013.354,185.283,369.681,166.930,55.693,160.269
C09738=1013.350,185.034,369.702,166.926,55.704,160.271
C09739=1013.346,184.785,369.723,166.922,55.716,160.272
C09740=1013.342,184.536,369.743,166.918,55.729,160.274
C09741=1013.339,184.286,369.764,166.913,55.741,160.275
C09742=1013.335,184.038,369.785,166.909,55.753,160.277
C09743=1013.331,183.788,369.806,166.905,55.764,160.278
C09744=1013.327,183.540,369.827,166.901,55.776,160.279
C09745=1013.324,183.290,369.847,166.897,55.789,160.281
C09746=1013.320,183.041,369.868,166.892,55.801,160.282
C09747=1013.316,182.792,369.889,166.889,55.813,160.284
C09748=1013.313,182.543,369.910,166.884,55.825,160.285
C09749=1013.309,182.293,369.931,166.880,55.837,160.287
C09750=1013.305,182.045,369.952,166.877,55.849,160.289
C09751=1013.301,181.795,369.972,166.873,55.861,160.290
C09752=1013.298,181.546,369.993,166.868,55.873,160.291
C09753=1013.293,181.297,370.014,166.864,55.885,160.293
C09754=1013.289,181.048,370.034,166.860,55.898,160.294
C09755=1013.285,180.798,370.054,166.856,55.909,160.296
C09756=1013.282,180.549,370.074,166.852,55.922,160.297
C09757=1013.277,180.301,370.094,166.848,55.934,160.299
C09758=1013.274,180.051,370.114,166.844,55.947,160.300
C09759=1013.269,179.801,370.134,166.839,55.959,160.302
C09760=1013.265,179.553,370.155,166.835,55.971,160.303
C09761=1013.261,179.303,370.175,166.831,55.983,160.305
C09762=1013.257,179.054,370.194,166.828,55.995,160.306
C09763=1013.253,178.805,370.214,166.824,56.008,160.308
C09764=1013.249,178.557,370.234,166.819,56.020,160.309
C09765=1013.245,178.307,370.254,166.815,56.032,160.311
C09766=1013.241,178.058,370.275,166.811,56.045,160.312
C09767=1013.236,177.808,370.294,166.807,56.056,160.314
C09768=1013.233,177.559,370.314,166.804,56.069,160.316
C09769=1013.228,177.310,370.335,166.799,56.081,160.317
C09770=1013.224,177.061,370.355,166.795,56.093,160.318
C09771=1013.220,176.812,370.374,166.792,56.105,160.320
C09772=1013.217,176.563,370.394,166.787,56.118,160.322
C09773=1013.213,176.313,370.414,166.783,56.130,160.323
C09774=1013.208,176.065,370.434,166.779,56.142,160.325
C09775=1013.205,175.815,370.455,166.776,56.154,160.326
C09776=1013.200,175.566,370.474,166.771,56.166,160.328
C09777=1013.197,175.317,370.494,166.767,56.179,160.329
C09778=1013.193,175.068,370.514,166.764,56.191,160.331
C09779=1013.189,174.819,370.534,166.760,56.203,160.332
C09780=1013.185,174.569,370.554,166.756,56.215,160.334
C09781=1013.181,174.320,370.573,166.752,56.227,160.335
C09782=1013.177,174.071,370.593,166.748,56.239,160.337
C09783=1013.173,173.822,370.614,166.744,56.251,160.338
C09784=1013.169,173.573,370.633,166.741,56.264,160.340
C09785=1013.165,173.324,370.654,166.736,56.276,160.341
C09786=1013.161,173.075,370.673,166.732,56.288,160.343
C09787=1013.157,172.825,370.693,166.729,56.299,160.344
C09788=1013.154,172.576,370.713,166.725,56.312,160.346
C09789=1013.149,172.327,370.733,166.722,56.324,160.347
C09790=1013.146,172.078,370.753,166.717,56.336,160.349
C09791=1013.141,171.829,370.772,166.713,56.348,160.350
C09792=1013.138,171.579,370.792,166.710,56.361,160.352
C09793=1013.133,171.330,370.812,166.706,56.373,160.353
C09794=1013.130,171.081,370.832,166.702,56.384,160.355
C09795=1013.126,170.802,370.854,166.698,56.398,160.357
C09796=1013.121,170.522,370.876,166.693,56.412,160.358
C09797=1013.117,170.244,370.898,166.690,56.425,160.360
C09798=1013.113,169.965,370.920,166.685,56.438,160.362
C09799=1013.109,169.715,370.940,166.681,56.451,160.363
C09800=1013.105,169.466,370.960,166.678,56.462,160.365
C09801=1013.101,169.217,370.979,166.674,56.475,160.366
C09802=1013.097,168.968,371.000,166.671,56.487,160.368
C09803=1013.093,168.719,371.019,166.666,56.499,160.369
C09804=1013.089,168.469,371.039,166.663,56.511,160.371
C09805=1013.086,168.220,371.059,166.660,56.522,160.372
C09806=1013.082,167.971,371.078,166.655,56.535,160.374
C09807=1013.079,167.722,371.098,166.652,56.546,160.375
C09808=1013.074,167.473,371.117,166.648,56.558,160.377
C09809=1013.071,167.223,371.137,166.645,56.570,160.378
C09810=1013.066,166.974,371.157,166.640,56.582,160.380
C09811=1013.063,166.725,371.177,166.638,56.595,160.382
C09812=1013.060,166.476,371.196,166.634,56.607,160.383
C09813=1013.056,166.227,371.215,166.630,56.619,160.385
C09814=1013.052,165.977,371.235,166.627,56.630,160.386
C09815=1013.048,165.728,371.255,166.623,56.643,160.388
C09816=1013.044,165.479,371.275,166.619,56.654,160.389
C09817=1013.041,165.229,371.295,166.616,56.666,160.391
C09818=1013.037,164.981,371.314,166.612,56.678,160.392
C09819=1013.034,164.731,371.333,166.609,56.690,160.394
C09820=1013.029,164.482,371.353,166.605,56.702,160.395
C09821=1013.026,164.233,371.373,166.601,56.714,160.397
C09822=1013.022,163.984,371.392,166.598,56.726,160.398
C09823=1013.019,163.734,371.411,166.595,56.737,160.400
C09824=1013.015,163.485,371.431,166.590,56.750,160.401
C09825=1013.011,163.236,371.451,166.587,56.761,160.403
C09826=1013.007,162.987,371.471,166.584,56.773,160.404
C09827=1013.004,162.738,371.489,166.581,56.785,160.406
C09828=1013.000,162.488,371.509,166.576,56.796,160.407
C09829=1012.996,162.239,371.529,166.573,56.808,160.409
C09830=1012.993,161.991,371.548,166.570,56.820,160.410
C09831=1012.989,161.741,371.568,166.566,56.832,160.412
C09832=1012.985,161.492,371.587,166.562,56.844,160.413
C09833=1012.981,161.242,371.607,166.559,56.856,160.415
C09834=1012.978,160.993,371.626,166.556,56.867,160.416
C09835=1012.974,160.744,371.646,166.553,56.879,160.418
C09836=1012.971,160.495,371.666,166.550,56.891,160.420
C09837=1012.967,160.246,371.684,166.545,56.903,160.421
C09838=1012.964,159.996,371.704,166.542,56.914,160.422
C09839=1012.959,159.747,371.724,166.539,56.926,160.424
C09840=1012.956,159.497,371.743,166.535,56.938,160.425
C09841=1012.952,159.249,371.762,166.532,56.950,160.427
C09842=1012.949,159.000,371.782,166.529,56.962,160.429
C09843=1012.945,158.750,371.802,166.525,56.973,160.430
C09844=1012.942,158.501,371.821,166.521,56.985,160.431
C09845=1012.938,158.251,371.840,166.518,56.997,160.433
C09846=1012.934,158.002,371.860,166.515,57.008,160.435
C09847=1012.930,157.753,371.878,166.512,57.020,160.436
C09848=1012.926,157.504,371.897,166.509,57.032,160.438
C09849=1012.923,157.254,371.917,166.505,57.044,160.439
C09850=1012.919,157.005,371.936,166.501,57.056,160.441
C09851=1012.915,156.756,371.954,166.498,57.068,160.442
C09852=1012.911,156.507,371.973,166.495,57.079,160.444
C09853=1012.908,156.258,371.992,166.491,57.091,160.445
C09854=1012.903,156.008,372.011,166.487,57.103,160.447
C09855=1012.899,155.759,372.030,166.484,57.115,160.448
C09856=1012.896,155.510,372.048,166.481,57.127,160.450
C09857=1012.892,155.260,372.067,166.478,57.139,160.451
C09858=1012.888,155.011,372.086,166.475,57.151,160.453
C09859=1012.883,154.732,372.108,166.471,57.164,160.455
C09860=1012.880,154.452,372.129,166.467,57.177,160.456
C09861=1012.875,154.173,372.150,166.463,57.190,160.458
C09862=1012.871,153.894,372.171,166.460,57.203,160.460
C09863=1012.868,153.645,372.189,166.457,57.215,160.461
C09864=1012.863,153.396,372.209,166.454,57.227,160.463
C09865=1012.859,153.146,372.228,166.451,57.239,160.465
C09866=1012.856,152.897,372.246,166.447,57.250,160.466
C09867=1012.852,152.647,372.265,166.443,57.262,160.467
C09868=1012.848,152.399,372.283,166.440,57.274,160.469
C09869=1012.844,152.149,372.302,166.437,57.286,160.471
C09870=1012.840,151.899,372.321,166.434,57.298,160.472
C09871=1012.837,151.651,372.340,166.431,57.309,160.474
C09872=1012.832,151.401,372.358,166.427,57.321,160.475
C09873=1012.829,151.152,372.377,166.424,57.332,160.477
C09874=1012.825,150.903,372.396,166.421,57.344,160.478
C09875=1012.822,150.654,372.414,166.418,57.356,160.480
C09876=1012.818,150.404,372.433,166.415,57.368,160.482
C09877=1012.814,150.155,372.451,166.411,57.379,160.483
C09878=1012.810,149.905,372.470,166.408,57.391,160.484
C09879=1012.807,149.656,372.488,166.405,57.403,160.486
C09880=1012.803,149.407,372.507,166.402,57.414,160.487
C09881=1012.799,149.158,372.525,166.399,57.426,160.489
C09882=1012.795,148.908,372.544,166.396,57.438,160.491
C09883=1012.791,148.659,372.562,166.393,57.450,160.492
C09884=1012.787,148.410,372.581,166.389,57.461,160.494
C09885=1012.783,148.161,372.599,166.386,57.473,160.495
C09886=1012.779,147.911,372.618,166.383,57.485,160.497
C09887=1012.776,147.662,372.636,166.380,57.496,160.498
C09888=1012.772,147.413,372.655,166.377,57.508,160.500
C09889=1012.768,147.164,372.673,166.373,57.519,160.501
C09890=1012.764,146.914,372.692,166.370,57.531,160.503
C09891=1012.761,146.665,372.711,166.368,57.542,160.505
C09892=1012.757,146.415,372.729,166.365,57.554,160.506
C09893=1012.753,146.167,372.747,166.362,57.565,160.508
C09894=1012.749,145.916,372.765,166.359,57.577,160.509
C09895=1012.746,145.667,372.784,166.355,57.589,160.511
C09896=1012.742,145.418,372.802,166.352,57.601,160.512
C09897=1012.738,145.169,372.821,166.349,57.612,160.513
C09898=1012.734,144.919,372.839,166.346,57.624,160.515
C09899=1012.730,144.670,372.857,166.344,57.635,160.517
C09900=1012.727,144.421,372.875,166.340,57.646,160.518
C09901=1012.723,144.171,372.894,166.337,57.658,160.520
C09902=1012.718,143.923,372.911,166.334,57.669,160.521
C09903=1012.714,143.673,372.930,166.331,57.681,160.523
C09904=1012.711,143.423,372.948,166.328,57.693,160.525
C09905=1012.707,143.175,372.966,166.324,57.705,160.526
C09906=1012.703,142.925,372.984,166.321,57.716,160.528
C09907=1012.700,142.675,373.002,166.319,57.727,160.529
C09908=1012.695,142.426,373.020,166.316,57.739,160.531
C09909=1012.692,142.177,373.039,166.313,57.750,160.532
C09910=1012.688,141.928,373.056,166.310,57.762,160.534
C09911=1012.684,141.678,373.074,166.306,57.774,160.535
C09912=1012.680,141.429,373.093,166.304,57.785,160.537
C09913=1012.676,141.179,373.110,166.301,57.796,160.538
C09914=1012.672,140.930,373.129,166.298,57.808,160.540
C09915=1012.669,140.681,373.147,166.294,57.820,160.541
C09916=1012.665,140.431,373.165,166.293,57.831,160.543
C09917=1012.661,140.182,373.183,166.289,57.842,160.544
C09918=1012.658,139.933,373.201,166.286,57.854,160.546
C09919=1012.653,139.683,373.219,166.284,57.865,160.548
C09920=1012.650,139.434,373.237,166.280,57.876,160.549
C09921=1012.646,139.186,373.256,166.278,57.888,160.551
C09922=1012.642,138.936,373.273,166.275,57.899,160.552
C09923=1012.638,138.638,373.295,166.271,57.913,160.554
C09924=1012.633,138.340,373.316,166.268,57.927,160.556
C09925=1012.628,138.042,373.338,166.265,57.940,160.558
C09926=1012.624,137.745,373.359,166.260,57.953,160.559
C09927=1012.621,137.495,373.377,166.259,57.965,160.561
C09928=1012.617,137.245,373.396,166.255,57.976,160.562
C09929=1012.613,136.996,373.413,166.252,57.987,160.564
C09930=1012.609,136.747,373.431,166.250,57.999,160.566
C09931=1012.605,136.497,373.449,166.247,58.010,160.567
C09932=1012.602,136.248,373.466,166.244,58.021,160.568
C09933=1012.598,135.999,373.484,166.241,58.033,160.570
C09934=1012.593,135.749,373.502,166.238,58.044,160.572
C09935=1012.590,135.500,373.520,166.236,58.055,160.573
C09936=1012.586,135.251,373.537,166.232,58.066,160.574
C09937=1012.582,135.002,373.555,166.230,58.078,160.576
C09938=1012.578,134.752,373.573,166.227,58.089,160.578
C09939=1012.546,148.398,372.188,166.347,57.641,160.519
C09940=1012.549,148.647,372.170,166.351,57.630,160.518
C09941=1012.553,148.897,372.151,166.353,57.619,160.516
C09942=1012.557,149.145,372.133,166.356,57.607,160.514
C09943=1012.561,149.395,372.114,166.359,57.596,160.513
C09944=1012.564,149.644,372.096,166.362,57.584,160.511
C09945=1012.569,149.893,372.077,166.366,57.572,160.510
C09946=1012.572,150.142,372.059,166.369,57.561,160.509
C09947=1012.576,150.392,372.040,166.372,57.549,160.507
C09948=1012.580,150.641,372.022,166.375,57.537,160.506
C09949=1012.584,150.891,372.003,166.378,57.526,160.504
C09950=1012.587,151.140,371.985,166.381,57.514,160.502
C09951=1012.591,151.389,371.966,166.385,57.502,160.501
C09952=1012.595,151.638,371.948,166.388,57.491,160.499
C09953=1012.598,151.887,371.929,166.391,57.479,160.498
C09954=1012.602,152.137,371.910,166.394,57.467,160.496
C09955=1012.606,152.386,371.892,166.397,57.456,160.495
C09956=1012.610,152.636,371.873,166.400,57.444,160.493
C09957=1012.613,152.884,371.855,166.404,57.433,160.492
C09958=1012.617,153.134,371.836,166.407,57.421,160.490
C09959=1012.621,153.384,371.817,166.410,57.409,160.489
C09960=1012.627,153.781,371.787,166.416,57.390,160.486
C09961=1012.633,154.179,371.758,166.421,57.372,160.484
C09962=1012.638,154.577,371.727,166.426,57.353,160.481
C09963=1012.644,154.976,371.697,166.431,57.334,160.479
C09964=1012.648,155.226,371.679,166.434,57.322,160.477
C09965=1012.652,155.474,371.659,166.437,57.311,160.476
C09966=1012.656,155.724,371.641,166.440,57.299,160.474
C09967=1012.660,155.972,371.622,166.445,57.287,160.473
C09968=1012.664,156.222,371.604,166.448,57.275,160.471
C09969=1012.667,156.471,371.585,166.451,57.263,160.470
C09970=1012.671,156.720,371.566,166.454,57.252,160.468
C09971=1012.676,156.970,371.547,166.457,57.240,160.467
C09972=1012.678,157.219,371.528,166.460,57.228,160.465
C09973=1012.682,157.469,371.509,166.465,57.216,160.464
C09974=1012.686,157.717,371.490,166.468,57.204,160.462
C09975=1012.690,157.967,371.471,166.471,57.193,160.461
C09976=1012.694,158.216,371.453,166.474,57.181,160.459
C09977=1012.697,158.465,371.433,166.477,57.169,160.457
C09978=1012.700,158.715,371.414,166.481,57.158,160.456
C09979=1012.705,158.964,371.394,166.485,57.145,160.455
C09980=1012.707,159.213,371.375,166.488,57.134,160.453
C09981=1012.712,159.462,371.356,166.491,57.122,160.451
C09982=1012.715,159.712,371.336,166.495,57.111,160.450
C09983=1012.719,159.961,371.317,166.498,57.099,160.449
C09984=1012.722,160.211,371.298,166.501,57.087,160.447
C09985=1012.726,160.460,371.278,166.504,57.075,160.445
C09986=1012.730,160.708,371.259,166.507,57.063,160.444
C09987=1012.733,160.958,371.239,166.512,57.052,160.443
C09988=1012.737,161.207,371.220,166.515,57.040,160.441
C09989=1012.740,161.457,371.201,166.518,57.028,160.439
C09990=1012.744,161.706,371.181,166.521,57.016,160.438
C09991=1012.747,161.954,371.162,166.524,57.005,160.436
C09992=1012.751,162.204,371.142,166.529,56.993,160.435
C09993=1012.755,162.453,371.123,166.532,56.981,160.434
C09994=1012.758,162.703,371.103,166.535,56.969,160.432
C09995=1012.762,162.952,371.084,166.539,56.958,160.430
C09996=1012.766,163.201,371.064,166.543,56.945,160.429
//INST
///DATE 2021/06/25 14:50
///ATTR SC,RW,RJ
////FRAME ROBOT
///GROUP1 RB1
NOP
MOVL C00000 V=800.0 PL=0
MOVL C00001 V=800.0 PL=0
MOVL C00002 V=800.0 PL=0
MOVL C00003 V=800.0 PL=0
MOVL C00004 V=800.0 PL=0
MOVL C00005 V=800.0 PL=0
MOVL C00006 V=800.0 PL=0
MOVL C00007 V=800.0 PL=0
MOVL C00008 V=800.0 PL=0
MOVL C00009 V=800.0 PL=0
MOVL C00010 V=800.0 PL=0
MOVL C00011 V=800.0 PL=0
MOVL C00012 V=800.0 PL=0
MOVL C00013 V=800.0 PL=0
MOVL C00014 V=800.0 PL=0
MOVL C00015 V=800.0 PL=0
MOVL C00016 V=800.0 PL=0
MOVL C00017 V=800.0 PL=0
MOVL C00018 V=800.0 PL=0
MOVL C00019 V=800.0 PL=0
MOVL C00020 V=800.0 PL=0
MOVL C00021 V=800.0 PL=0
MOVL C00022 V=800.0 PL=0
MOVL C00023 V=800.0 PL=0
MOVL C00024 V=800.0 PL=0
MOVL C00025 V=800.0 PL=0
MOVL C00026 V=800.0 PL=0
MOVL C00027 V=800.0 PL=0
MOVL C00028 V=800.0 PL=0
MOVL C00029 V=800.0 PL=0
MOVL C00030 V=800.0 PL=0
MOVL C00031 V=800.0 PL=0
MOVL C00032 V=800.0 PL=0
MOVL C00033 V=800.0 PL=0
MOVL C00034 V=800.0 PL=0
MOVL C00035 V=800.0 PL=0
MOVL C00036 V=800.0 PL=0
MOVL C00037 V=800.0 PL=0
MOVL C00038 V=800.0 PL=0
MOVL C00039 V=800.0 PL=0
MOVL C00040 V=800.0 PL=0
MOVL C00041 V=800.0 PL=0
MOVL C00042 V=800.0 PL=0
MOVL C00043 V=800.0 PL=0
MOVL C00044 V=800.0 PL=0
MOVL C00045 V=800.0 PL=0
MOVL C00046 V=800.0 PL=0
MOVL C00047 V=800.0 PL=0
MOVL C00048 V=800.0 PL=0
MOVL C00049 V=800.0 PL=0
MOVL C00050 V=800.0 PL=0
MOVL C00051 V=800.0 PL=0
MOVL C00052 V=800.0 PL=0
MOVL C00053 V=800.0 PL=0
MOVL C00054 V=800.0 PL=0
MOVL C00055 V=800.0 PL=0
MOVL C00056 V=800.0 PL=0
MOVL C00057 V=800.0 PL=0
MOVL C00058 V=800.0 PL=0
MOVL C00059 V=800.0 PL=0
MOVL C00060 V=800.0 PL=0
MOVL C00061 V=800.0 PL=0
MOVL C00062 V=800.0 PL=0
MOVL C00063 V=800.0 PL=0
MOVL C00064 V=800.0 PL=0
MOVL C00065 V=800.0 PL=0
MOVL C00066 V=800.0 PL=0
MOVL C00067 V=800.0 PL=0
MOVL C00068 V=800.0 PL=0
MOVL C00069 V=800.0 PL=0
MOVL C00070 V=800.0 PL=0
MOVL C00071 V=800.0 PL=0
MOVL C00072 V=800.0 PL=0
MOVL C00073 V=800.0 PL=0
MOVL C00074 V=800.0 PL=0
MOVL C00075 V=800.0 PL=0
MOVL C00076 V=800.0 PL=0
MOVL C00077 V=800.0 PL=0
MOVL C00078 V=800.0 PL=0
MOVL C00079 V=800.0 PL=0
MOVL C00080 V=800.0 PL=0
MOVL C00081 V=800.0 PL=0
MOVL C00082 V=800.0 PL=0
MOVL C00083 V=800.0 PL=0
MOVL C00084 V=800.0 PL=0
MOVL C00085 V=800.0 PL=0
MOVL C00086 V=800.0 PL=0
MOVL C00087 V=800.0 PL=0
MOVL C00088 V=800.0 PL=0
MOVL C00089 V=800.0 PL=0
MOVL C00090 V=800.0 PL=0
MOVL C00091 V=800.0 PL=0
MOVL C00092 V=800.0 PL=0
MOVL C00093 V=800.0 PL=0
MOVL C00094 V=800.0 PL=0
MOVL C00095 V=800.0 PL=0
MOVL C00096 V=800.0 PL=0
MOVL C00097 V=800.0 PL=0
MOVL C00098 V=800.0 PL=0
MOVL C00099 V=800.0 PL=0
MOVL C00100 V=800.0 PL=0
MOVL C00101 V=800.0 PL=0
MOVL C00102 V=800.0 PL=0
MOVL C00103 V=800.0 PL=0
MOVL C00104 V=800.0 PL=0
MOVL C00105 V=800.0 PL=0
MOVL C00106 V=800.0 PL=0
MOVL C00107 V=800.0 PL=0
MOVL C00108 V=800.0 PL=0
MOVL C00109 V=800.0 PL=0
MOVL C00110 V=800.0 PL=0
MOVL C00111 V=800.0 PL=0
MOVL C00112 V=800.0 PL=0
MOVL C00113 V=800.0 PL=0
MOVL C00114 V=800.0 PL=0
MOVL C00115 V=800.0 PL=0
MOVL C00116 V=800.0 PL=0
MOVL C00117 V=800.0 PL=0
MOVL C00118 V=800.0 PL=0
MOVL C00119 V=800.0 PL=0
MOVL C00120 V=800.0 PL=0
MOVL C00121 V=800.0 PL=0
MOVL C00122 V=800.0 PL=0
MOVL C00123 V=800.0 PL=0
MOVL C00124 V=800.0 PL=0
MOVL C00125 V=800.0 PL=0
MOVL C00126 V=800.0 PL=0
MOVL C00127 V=800.0 PL=0
MOVL C00128 V=800.0 PL=0
MOVL C00129 V=800.0 PL=0
MOVL C00130 V=800.0 PL=0
MOVL C00131 V=800.0 PL=0
MOVL C00132 V=800.0 PL=0
MOVL C00133 V=800.0 PL=0
MOVL C00134 V=800.0 PL=0
MOVL C00135 V=800.0 PL=0
MOVL C00136 V=800.0 PL=0
MOVL C00137 V=800.0 PL=0
MOVL C00138 V=800.0 PL=0
MOVL C00139 V=800.0 PL=0
MOVL C00140 V=800.0 PL=0
MOVL C00141 V=800.0 PL=0
MOVL C00142 V=800.0 PL=0
MOVL C00143 V=800.0 PL=0
MOVL C00144 V=800.0 PL=0
MOVL C00145 V=800.0 PL=0
MOVL C00146 V=800.0 PL=0
MOVL C00147 V=800.0 PL=0
MOVL C00148 V=800.0 PL=0
MOVL C00149 V=800.0 PL=0
MOVL C00150 V=800.0 PL=0
MOVL C00151 V=800.0 PL=0
MOVL C00152 V=800.0 PL=0
MOVL C00153 V=800.0 PL=0
MOVL C00154 V=800.0 PL=0
MOVL C00155 V=800.0 PL=0
MOVL C00156 V=800.0 PL=0
MOVL C00157 V=800.0 PL=0
MOVL C00158 V=800.0 PL=0
MOVL C00159 V=800.0 PL=0
MOVL C00160 V=800.0 PL=0
MOVL C00161 V=800.0 PL=0
MOVL C00162 V=800.0 PL=0
MOVL C00163 V=800.0 PL=0
MOVL C00164 V=800.0 PL=0
MOVL C00165 V=800.0 PL=0
MOVL C00166 V=800.0 PL=0
MOVL C00167 V=800.0 PL=0
MOVL C00168 V=800.0 PL=0
MOVL C00169 V=800.0 PL=0
MOVL C00170 V=800.0 PL=0
MOVL C00171 V=800.0 PL=0
MOVL C00172 V=800.0 PL=0
MOVL C00173 V=800.0 PL=0
MOVL C00174 V=800.0 PL=0
MOVL C00175 V=800.0 PL=0
MOVL C00176 V=800.0 PL=0
MOVL C00177 V=800.0 PL=0
MOVL C00178 V=800.0 PL=0
MOVL C00179 V=800.0 PL=0
MOVL C00180 V=800.0 PL=0
MOVL C00181 V=800.0 PL=0
MOVL C00182 V=800.0 PL=0
MOVL C00183 V=800.0 PL=0
MOVL C00184 V=800.0 PL=0
MOVL C00185 V=800.0 PL=0
MOVL C00186 V=800.0 PL=0
MOVL C00187 V=800.0 PL=0
MOVL C00188 V=800.0 PL=0
MOVL C00189 V=800.0 PL=0
MOVL C00190 V=800.0 PL=0
MOVL C00191 V=800.0 PL=0
MOVL C00192 V=800.0 PL=0
MOVL C00193 V=800.0 PL=0
MOVL C00194 V=800.0 PL=0
MOVL C00195 V=800.0 PL=0
MOVL C00196 V=800.0 PL=0
MOVL C00197 V=800.0 PL=0
MOVL C00198 V=800.0 PL=0
MOVL C00199 V=800.0 PL=0
MOVL C00200 V=800.0 PL=0
MOVL C00201 V=800.0 PL=0
MOVL C00202 V=800.0 PL=0
MOVL C00203 V=800.0 PL=0
MOVL C00204 V=800.0 PL=0
MOVL C00205 V=800.0 PL=0
MOVL C00206 V=800.0 PL=0
MOVL C00207 V=800.0 PL=0
MOVL C00208 V=800.0 PL=0
MOVL C00209 V=800.0 PL=0
MOVL C00210 V=800.0 PL=0
MOVL C00211 V=800.0 PL=0
MOVL C00212 V=800.0 PL=0
MOVL C00213 V=800.0 PL=0
MOVL C00214 V=800.0 PL=0
MOVL C00215 V=800.0 PL=0
MOVL C00216 V=800.0 PL=0
MOVL C00217 V=800.0 PL=0
MOVL C00218 V=800.0 PL=0
MOVL C00219 V=800.0 PL=0
MOVL C00220 V=800.0 PL=0
MOVL C00221 V=800.0 PL=0
MOVL C00222 V=800.0 PL=0
MOVL C00223 V=800.0 PL=0
MOVL C00224 V=800.0 PL=0
MOVL C00225 V=800.0 PL=0
MOVL C00226 V=800.0 PL=0
MOVL C00227 V=800.0 PL=0
MOVL C00228 V=800.0 PL=0
MOVL C00229 V=800.0 PL=0
MOVL C00230 V=800.0 PL=0
MOVL C00231 V=800.0 PL=0
MOVL C00232 V=800.0 PL=0
MOVL C00233 V=800.0 PL=0
MOVL C00234 V=800.0 PL=0
MOVL C00235 V=800.0 PL=0
MOVL C00236 V=800.0 PL=0
MOVL C00237 V=800.0 PL=0
MOVL C00238 V=800.0 PL=0
MOVL C00239 V=800.0 PL=0
MOVL C00240 V=800.0 PL=0
MOVL C00241 V=800.0 PL=0
MOVL C00242 V=800.0 PL=0
MOVL C00243 V=800.0 PL=0
MOVL C00244 V=800.0 PL=0
MOVL C00245 V=800.0 PL=0
MOVL C00246 V=800.0 PL=0
MOVL C00247 V=800.0 PL=0
MOVL C00248 V=800.0 PL=0
MOVL C00249 V=800.0 PL=0
MOVL C00250 V=800.0 PL=0
MOVL C00251 V=800.0 PL=0
MOVL C00252 V=800.0 PL=0
MOVL C00253 V=800.0 PL=0
MOVL C00254 V=800.0 PL=0
MOVL C00255 V=800.0 PL=0
MOVL C00256 V=800.0 PL=0
MOVL C00257 V=800.0 PL=0
MOVL C00258 V=800.0 PL=0
MOVL C00259 V=800.0 PL=0
MOVL C00260 V=800.0 PL=0
MOVL C00261 V=800.0 PL=0
MOVL C00262 V=800.0 PL=0
MOVL C00263 V=800.0 PL=0
MOVL C00264 V=800.0 PL=0
MOVL C00265 V=800.0 PL=0
MOVL C00266 V=800.0 PL=0
MOVL C00267 V=800.0 PL=0
MOVL C00268 V=800.0 PL=0
MOVL C00269 V=800.0 PL=0
MOVL C00270 V=800.0 PL=0
MOVL C00271 V=800.0 PL=0
MOVL C00272 V=800.0 PL=0
MOVL C00273 V=800.0 PL=0
MOVL C00274 V=800.0 PL=0
MOVL C00275 V=800.0 PL=0
MOVL C00276 V=800.0 PL=0
MOVL C00277 V=800.0 PL=0
MOVL C00278 V=800.0 PL=0
MOVL C00279 V=800.0 PL=0
MOVL C00280 V=800.0 PL=0
MOVL C00281 V=800.0 PL=0
MOVL C00282 V=800.0 PL=0
MOVL C00283 V=800.0 PL=0
MOVL C00284 V=800.0 PL=0
MOVL C00285 V=800.0 PL=0
MOVL C00286 V=800.0 PL=0
MOVL C00287 V=800.0 PL=0
MOVL C00288 V=800.0 PL=0
MOVL C00289 V=800.0 PL=0
MOVL C00290 V=800.0 PL=0
MOVL C00291 V=800.0 PL=0
MOVL C00292 V=800.0 PL=0
MOVL C00293 V=800.0 PL=0
MOVL C00294 V=800.0 PL=0
MOVL C00295 V=800.0 PL=0
MOVL C00296 V=800.0 PL=0
MOVL C00297 V=800.0 PL=0
MOVL C00298 V=800.0 PL=0
MOVL C00299 V=800.0 PL=0
MOVL C00300 V=800.0 PL=0
MOVL C00301 V=800.0 PL=0
MOVL C00302 V=800.0 PL=0
MOVL C00303 V=800.0 PL=0
MOVL C00304 V=800.0 PL=0
MOVL C00305 V=800.0 PL=0
MOVL C00306 V=800.0 PL=0
MOVL C00307 V=800.0 PL=0
MOVL C00308 V=800.0 PL=0
MOVL C00309 V=800.0 PL=0
MOVL C00310 V=800.0 PL=0
MOVL C00311 V=800.0 PL=0
MOVL C00312 V=800.0 PL=0
MOVL C00313 V=800.0 PL=0
MOVL C00314 V=800.0 PL=0
MOVL C00315 V=800.0 PL=0
MOVL C00316 V=800.0 PL=0
MOVL C00317 V=800.0 PL=0
MOVL C00318 V=800.0 PL=0
MOVL C00319 V=800.0 PL=0
MOVL C00320 V=800.0 PL=0
MOVL C00321 V=800.0 PL=0
MOVL C00322 V=800.0 PL=0
MOVL C00323 V=800.0 PL=0
MOVL C00324 V=800.0 PL=0
MOVL C00325 V=800.0 PL=0
MOVL C00326 V=800.0 PL=0
MOVL C00327 V=800.0 PL=0
MOVL C00328 V=800.0 PL=0
MOVL C00329 V=800.0 PL=0
MOVL C00330 V=800.0 PL=0
MOVL C00331 V=800.0 PL=0
MOVL C00332 V=800.0 PL=0
MOVL C00333 V=800.0 PL=0
MOVL C00334 V=800.0 PL=0
MOVL C00335 V=800.0 PL=0
MOVL C00336 V=800.0 PL=0
MOVL C00337 V=800.0 PL=0
MOVL C00338 V=800.0 PL=0
MOVL C00339 V=800.0 PL=0
MOVL C00340 V=800.0 PL=0
MOVL C00341 V=800.0 PL=0
MOVL C00342 V=800.0 PL=0
MOVL C00343 V=800.0 PL=0
MOVL C00344 V=800.0 PL=0
MOVL C00345 V=800.0 PL=0
MOVL C00346 V=800.0 PL=0
MOVL C00347 V=800.0 PL=0
MOVL C00348 V=800.0 PL=0
MOVL C00349 V=800.0 PL=0
MOVL C00350 V=800.0 PL=0
MOVL C00351 V=800.0 PL=0
MOVL C00352 V=800.0 PL=0
MOVL C00353 V=800.0 PL=0
MOVL C00354 V=800.0 PL=0
MOVL C00355 V=800.0 PL=0
MOVL C00356 V=800.0 PL=0
MOVL C00357 V=800.0 PL=0
MOVL C00358 V=800.0 PL=0
MOVL C00359 V=800.0 PL=0
MOVL C00360 V=800.0 PL=0
MOVL C00361 V=800.0 PL=0
MOVL C00362 V=800.0 PL=0
MOVL C00363 V=800.0 PL=0
MOVL C00364 V=800.0 PL=0
MOVL C00365 V=800.0 PL=0
MOVL C00366 V=800.0 PL=0
MOVL C00367 V=800.0 PL=0
MOVL C00368 V=800.0 PL=0
MOVL C00369 V=800.0 PL=0
MOVL C00370 V=800.0 PL=0
MOVL C00371 V=800.0 PL=0
MOVL C00372 V=800.0 PL=0
MOVL C00373 V=800.0 PL=0
MOVL C00374 V=800.0 PL=0
MOVL C00375 V=800.0 PL=0
MOVL C00376 V=800.0 PL=0
MOVL C00377 V=800.0 PL=0
MOVL C00378 V=800.0 PL=0
MOVL C00379 V=800.0 PL=0
MOVL C00380 V=800.0 PL=0
MOVL C00381 V=800.0 PL=0
MOVL C00382 V=800.0 PL=0
MOVL C00383 V=800.0 PL=0
MOVL C00384 V=800.0 PL=0
MOVL C00385 V=800.0 PL=0
MOVL C00386 V=800.0 PL=0
MOVL C00387 V=800.0 PL=0
MOVL C00388 V=800.0 PL=0
MOVL C00389 V=800.0 PL=0
MOVL C00390 V=800.0 PL=0
MOVL C00391 V=800.0 PL=0
MOVL C00392 V=800.0 PL=0
MOVL C00393 V=800.0 PL=0
MOVL C00394 V=800.0 PL=0
MOVL C00395 V=800.0 PL=0
MOVL C00396 V=800.0 PL=0
MOVL C00397 V=800.0 PL=0
MOVL C00398 V=800.0 PL=0
MOVL C00399 V=800.0 PL=0
MOVL C00400 V=800.0 PL=0
MOVL C00401 V=800.0 PL=0
MOVL C00402 V=800.0 PL=0
MOVL C00403 V=800.0 PL=0
MOVL C00404 V=800.0 PL=0
MOVL C00405 V=800.0 PL=0
MOVL C00406 V=800.0 PL=0
MOVL C00407 V=800.0 PL=0
MOVL C00408 V=800.0 PL=0
MOVL C00409 V=800.0 PL=0
MOVL C00410 V=800.0 PL=0
MOVL C00411 V=800.0 PL=0
MOVL C00412 V=800.0 PL=0
MOVL C00413 V=800.0 PL=0
MOVL C00414 V=800.0 PL=0
MOVL C00415 V=800.0 PL=0
MOVL C00416 V=800.0 PL=0
MOVL C00417 V=800.0 PL=0
MOVL C00418 V=800.0 PL=0
MOVL C00419 V=800.0 PL=0
MOVL C00420 V=800.0 PL=0
MOVL C00421 V=800.0 PL=0
MOVL C00422 V=800.0 PL=0
MOVL C00423 V=800.0 PL=0
MOVL C00424 V=800.0 PL=0
MOVL C00425 V=800.0 PL=0
MOVL C00426 V=800.0 PL=0
MOVL C00427 V=800.0 PL=0
MOVL C00428 V=800.0 PL=0
MOVL C00429 V=800.0 PL=0
MOVL C00430 V=800.0 PL=0
MOVL C00431 V=800.0 PL=0
MOVL C00432 V=800.0 PL=0
MOVL C00433 V=800.0 PL=0
MOVL C00434 V=800.0 PL=0
MOVL C00435 V=800.0 PL=0
MOVL C00436 V=800.0 PL=0
MOVL C00437 V=800.0 PL=0
MOVL C00438 V=800.0 PL=0
MOVL C00439 V=800.0 PL=0
MOVL C00440 V=800.0 PL=0
MOVL C00441 V=800.0 PL=0
MOVL C00442 V=800.0 PL=0
MOVL C00443 V=800.0 PL=0
MOVL C00444 V=800.0 PL=0
MOVL C00445 V=800.0 PL=0
MOVL C00446 V=800.0 PL=0
MOVL C00447 V=800.0 PL=0
MOVL C00448 V=800.0 PL=0
MOVL C00449 V=800.0 PL=0
MOVL C00450 V=800.0 PL=0
MOVL C00451 V=800.0 PL=0
MOVL C00452 V=800.0 PL=0
MOVL C00453 V=800.0 PL=0
MOVL C00454 V=800.0 PL=0
MOVL C00455 V=800.0 PL=0
MOVL C00456 V=800.0 PL=0
MOVL C00457 V=800.0 PL=0
MOVL C00458 V=800.0 PL=0
MOVL C00459 V=800.0 PL=0
MOVL C00460 V=800.0 PL=0
MOVL C00461 V=800.0 PL=0
MOVL C00462 V=800.0 PL=0
MOVL C00463 V=800.0 PL=0
MOVL C00464 V=800.0 PL=0
MOVL C00465 V=800.0 PL=0
MOVL C00466 V=800.0 PL=0
MOVL C00467 V=800.0 PL=0
MOVL C00468 V=800.0 PL=0
MOVL C00469 V=800.0 PL=0
MOVL C00470 V=800.0 PL=0
MOVL C00471 V=800.0 PL=0
MOVL C00472 V=800.0 PL=0
MOVL C00473 V=800.0 PL=0
MOVL C00474 V=800.0 PL=0
MOVL C00475 V=800.0 PL=0
MOVL C00476 V=800.0 PL=0
MOVL C00477 V=800.0 PL=0
MOVL C00478 V=800.0 PL=0
MOVL C00479 V=800.0 PL=0
MOVL C00480 V=800.0 PL=0
MOVL C00481 V=800.0 PL=0
MOVL C00482 V=800.0 PL=0
MOVL C00483 V=800.0 PL=0
MOVL C00484 V=800.0 PL=0
MOVL C00485 V=800.0 PL=0
MOVL C00486 V=800.0 PL=0
MOVL C00487 V=800.0 PL=0
MOVL C00488 V=800.0 PL=0
MOVL C00489 V=800.0 PL=0
MOVL C00490 V=800.0 PL=0
MOVL C00491 V=800.0 PL=0
MOVL C00492 V=800.0 PL=0
MOVL C00493 V=800.0 PL=0
MOVL C00494 V=800.0 PL=0
MOVL C00495 V=800.0 PL=0
MOVL C00496 V=800.0 PL=0
MOVL C00497 V=800.0 PL=0
MOVL C00498 V=800.0 PL=0
MOVL C00499 V=800.0 PL=0
MOVL C00500 V=800.0 PL=0
MOVL C00501 V=800.0 PL=0
MOVL C00502 V=800.0 PL=0
MOVL C00503 V=800.0 PL=0
MOVL C00504 V=800.0 PL=0
MOVL C00505 V=800.0 PL=0
MOVL C00506 V=800.0 PL=0
MOVL C00507 V=800.0 PL=0
MOVL C00508 V=800.0 PL=0
MOVL C00509 V=800.0 PL=0
MOVL C00510 V=800.0 PL=0
MOVL C00511 V=800.0 PL=0
MOVL C00512 V=800.0 PL=0
MOVL C00513 V=800.0 PL=0
MOVL C00514 V=800.0 PL=0
MOVL C00515 V=800.0 PL=0
MOVL C00516 V=800.0 PL=0
MOVL C00517 V=800.0 PL=0
MOVL C00518 V=800.0 PL=0
MOVL C00519 V=800.0 PL=0
MOVL C00520 V=800.0 PL=0
MOVL C00521 V=800.0 PL=0
MOVL C00522 V=800.0 PL=0
MOVL C00523 V=800.0 PL=0
MOVL C00524 V=800.0 PL=0
MOVL C00525 V=800.0 PL=0
MOVL C00526 V=800.0 PL=0
MOVL C00527 V=800.0 PL=0
MOVL C00528 V=800.0 PL=0
MOVL C00529 V=800.0 PL=0
MOVL C00530 V=800.0 PL=0
MOVL C00531 V=800.0 PL=0
MOVL C00532 V=800.0 PL=0
MOVL C00533 V=800.0 PL=0
MOVL C00534 V=800.0 PL=0
MOVL C00535 V=800.0 PL=0
MOVL C00536 V=800.0 PL=0
MOVL C00537 V=800.0 PL=0
MOVL C00538 V=800.0 PL=0
MOVL C00539 V=800.0 PL=0
MOVL C00540 V=800.0 PL=0
MOVL C00541 V=800.0 PL=0
MOVL C00542 V=800.0 PL=0
MOVL C00543 V=800.0 PL=0
MOVL C00544 V=800.0 PL=0
MOVL C00545 V=800.0 PL=0
MOVL C00546 V=800.0 PL=0
MOVL C00547 V=800.0 PL=0
MOVL C00548 V=800.0 PL=0
MOVL C00549 V=800.0 PL=0
MOVL C00550 V=800.0 PL=0
MOVL C00551 V=800.0 PL=0
MOVL C00552 V=800.0 PL=0
MOVL C00553 V=800.0 PL=0
MOVL C00554 V=800.0 PL=0
MOVL C00555 V=800.0 PL=0
MOVL C00556 V=800.0 PL=0
MOVL C00557 V=800.0 PL=0
MOVL C00558 V=800.0 PL=0
MOVL C00559 V=800.0 PL=0
MOVL C00560 V=800.0 PL=0
MOVL C00561 V=800.0 PL=0
MOVL C00562 V=800.0 PL=0
MOVL C00563 V=800.0 PL=0
MOVL C00564 V=800.0 PL=0
MOVL C00565 V=800.0 PL=0
MOVL C00566 V=800.0 PL=0
MOVL C00567 V=800.0 PL=0
MOVL C00568 V=800.0 PL=0
MOVL C00569 V=800.0 PL=0
MOVL C00570 V=800.0 PL=0
MOVL C00571 V=800.0 PL=0
MOVL C00572 V=800.0 PL=0
MOVL C00573 V=800.0 PL=0
MOVL C00574 V=800.0 PL=0
MOVL C00575 V=800.0 PL=0
MOVL C00576 V=800.0 PL=0
MOVL C00577 V=800.0 PL=0
MOVL C00578 V=800.0 PL=0
MOVL C00579 V=800.0 PL=0
MOVL C00580 V=800.0 PL=0
MOVL C00581 V=800.0 PL=0
MOVL C00582 V=800.0 PL=0
MOVL C00583 V=800.0 PL=0
MOVL C00584 V=800.0 PL=0
MOVL C00585 V=800.0 PL=0
MOVL C00586 V=800.0 PL=0
MOVL C00587 V=800.0 PL=0
MOVL C00588 V=800.0 PL=0
MOVL C00589 V=800.0 PL=0
MOVL C00590 V=800.0 PL=0
MOVL C00591 V=800.0 PL=0
MOVL C00592 V=800.0 PL=0
MOVL C00593 V=800.0 PL=0
MOVL C00594 V=800.0 PL=0
MOVL C00595 V=800.0 PL=0
MOVL C00596 V=800.0 PL=0
MOVL C00597 V=800.0 PL=0
MOVL C00598 V=800.0 PL=0
MOVL C00599 V=800.0 PL=0
MOVL C00600 V=800.0 PL=0
MOVL C00601 V=800.0 PL=0
MOVL C00602 V=800.0 PL=0
MOVL C00603 V=800.0 PL=0
MOVL C00604 V=800.0 PL=0
MOVL C00605 V=800.0 PL=0
MOVL C00606 V=800.0 PL=0
MOVL C00607 V=800.0 PL=0
MOVL C00608 V=800.0 PL=0
MOVL C00609 V=800.0 PL=0
MOVL C00610 V=800.0 PL=0
MOVL C00611 V=800.0 PL=0
MOVL C00612 V=800.0 PL=0
MOVL C00613 V=800.0 PL=0
MOVL C00614 V=800.0 PL=0
MOVL C00615 V=800.0 PL=0
MOVL C00616 V=800.0 PL=0
MOVL C00617 V=800.0 PL=0
MOVL C00618 V=800.0 PL=0
MOVL C00619 V=800.0 PL=0
MOVL C00620 V=800.0 PL=0
MOVL C00621 V=800.0 PL=0
MOVL C00622 V=800.0 PL=0
MOVL C00623 V=800.0 PL=0
MOVL C00624 V=800.0 PL=0
MOVL C00625 V=800.0 PL=0
MOVL C00626 V=800.0 PL=0
MOVL C00627 V=800.0 PL=0
MOVL C00628 V=800.0 PL=0
MOVL C00629 V=800.0 PL=0
MOVL C00630 V=800.0 PL=0
MOVL C00631 V=800.0 PL=0
MOVL C00632 V=800.0 PL=0
MOVL C00633 V=800.0 PL=0
MOVL C00634 V=800.0 PL=0
MOVL C00635 V=800.0 PL=0
MOVL C00636 V=800.0 PL=0
MOVL C00637 V=800.0 PL=0
MOVL C00638 V=800.0 PL=0
MOVL C00639 V=800.0 PL=0
MOVL C00640 V=800.0 PL=0
MOVL C00641 V=800.0 PL=0
MOVL C00642 V=800.0 PL=0
MOVL C00643 V=800.0 PL=0
MOVL C00644 V=800.0 PL=0
MOVL C00645 V=800.0 PL=0
MOVL C00646 V=800.0 PL=0
MOVL C00647 V=800.0 PL=0
MOVL C00648 V=800.0 PL=0
MOVL C00649 V=800.0 PL=0
MOVL C00650 V=800.0 PL=0
MOVL C00651 V=800.0 PL=0
MOVL C00652 V=800.0 PL=0
MOVL C00653 V=800.0 PL=0
MOVL C00654 V=800.0 PL=0
MOVL C00655 V=800.0 PL=0
MOVL C00656 V=800.0 PL=0
MOVL C00657 V=800.0 PL=0
MOVL C00658 V=800.0 PL=0
MOVL C00659 V=800.0 PL=0
MOVL C00660 V=800.0 PL=0
MOVL C00661 V=800.0 PL=0
MOVL C00662 V=800.0 PL=0
MOVL C00663 V=800.0 PL=0
MOVL C00664 V=800.0 PL=0
MOVL C00665 V=800.0 PL=0
MOVL C00666 V=800.0 PL=0
MOVL C00667 V=800.0 PL=0
MOVL C00668 V=800.0 PL=0
MOVL C00669 V=800.0 PL=0
MOVL C00670 V=800.0 PL=0
MOVL C00671 V=800.0 PL=0
MOVL C00672 V=800.0 PL=0
MOVL C00673 V=800.0 PL=0
MOVL C00674 V=800.0 PL=0
MOVL C00675 V=800.0 PL=0
MOVL C00676 V=800.0 PL=0
MOVL C00677 V=800.0 PL=0
MOVL C00678 V=800.0 PL=0
MOVL C00679 V=800.0 PL=0
MOVL C00680 V=800.0 PL=0
MOVL C00681 V=800.0 PL=0
MOVL C00682 V=800.0 PL=0
MOVL C00683 V=800.0 PL=0
MOVL C00684 V=800.0 PL=0
MOVL C00685 V=800.0 PL=0
MOVL C00686 V=800.0 PL=0
MOVL C00687 V=800.0 PL=0
MOVL C00688 V=800.0 PL=0
MOVL C00689 V=800.0 PL=0
MOVL C00690 V=800.0 PL=0
MOVL C00691 V=800.0 PL=0
MOVL C00692 V=800.0 PL=0
MOVL C00693 V=800.0 PL=0
MOVL C00694 V=800.0 PL=0
MOVL C00695 V=800.0 PL=0
MOVL C00696 V=800.0 PL=0
MOVL C00697 V=800.0 PL=0
MOVL C00698 V=800.0 PL=0
MOVL C00699 V=800.0 PL=0
MOVL C00700 V=800.0 PL=0
MOVL C00701 V=800.0 PL=0
MOVL C00702 V=800.0 PL=0
MOVL C00703 V=800.0 PL=0
MOVL C00704 V=800.0 PL=0
MOVL C00705 V=800.0 PL=0
MOVL C00706 V=800.0 PL=0
MOVL C00707 V=800.0 PL=0
MOVL C00708 V=800.0 PL=0
MOVL C00709 V=800.0 PL=0
MOVL C00710 V=800.0 PL=0
MOVL C00711 V=800.0 PL=0
MOVL C00712 V=800.0 PL=0
MOVL C00713 V=800.0 PL=0
MOVL C00714 V=800.0 PL=0
MOVL C00715 V=800.0 PL=0
MOVL C00716 V=800.0 PL=0
MOVL C00717 V=800.0 PL=0
MOVL C00718 V=800.0 PL=0
MOVL C00719 V=800.0 PL=0
MOVL C00720 V=800.0 PL=0
MOVL C00721 V=800.0 PL=0
MOVL C00722 V=800.0 PL=0
MOVL C00723 V=800.0 PL=0
MOVL C00724 V=800.0 PL=0
MOVL C00725 V=800.0 PL=0
MOVL C00726 V=800.0 PL=0
MOVL C00727 V=800.0 PL=0
MOVL C00728 V=800.0 PL=0
MOVL C00729 V=800.0 PL=0
MOVL C00730 V=800.0 PL=0
MOVL C00731 V=800.0 PL=0
MOVL C00732 V=800.0 PL=0
MOVL C00733 V=800.0 PL=0
MOVL C00734 V=800.0 PL=0
MOVL C00735 V=800.0 PL=0
MOVL C00736 V=800.0 PL=0
MOVL C00737 V=800.0 PL=0
MOVL C00738 V=800.0 PL=0
MOVL C00739 V=800.0 PL=0
MOVL C00740 V=800.0 PL=0
MOVL C00741 V=800.0 PL=0
MOVL C00742 V=800.0 PL=0
MOVL C00743 V=800.0 PL=0
MOVL C00744 V=800.0 PL=0
MOVL C00745 V=800.0 PL=0
MOVL C00746 V=800.0 PL=0
MOVL C00747 V=800.0 PL=0
MOVL C00748 V=800.0 PL=0
MOVL C00749 V=800.0 PL=0
MOVL C00750 V=800.0 PL=0
MOVL C00751 V=800.0 PL=0
MOVL C00752 V=800.0 PL=0
MOVL C00753 V=800.0 PL=0
MOVL C00754 V=800.0 PL=0
MOVL C00755 V=800.0 PL=0
MOVL C00756 V=800.0 PL=0
MOVL C00757 V=800.0 PL=0
MOVL C00758 V=800.0 PL=0
MOVL C00759 V=800.0 PL=0
MOVL C00760 V=800.0 PL=0
MOVL C00761 V=800.0 PL=0
MOVL C00762 V=800.0 PL=0
MOVL C00763 V=800.0 PL=0
MOVL C00764 V=800.0 PL=0
MOVL C00765 V=800.0 PL=0
MOVL C00766 V=800.0 PL=0
MOVL C00767 V=800.0 PL=0
MOVL C00768 V=800.0 PL=0
MOVL C00769 V=800.0 PL=0
MOVL C00770 V=800.0 PL=0
MOVL C00771 V=800.0 PL=0
MOVL C00772 V=800.0 PL=0
MOVL C00773 V=800.0 PL=0
MOVL C00774 V=800.0 PL=0
MOVL C00775 V=800.0 PL=0
MOVL C00776 V=800.0 PL=0
MOVL C00777 V=800.0 PL=0
MOVL C00778 V=800.0 PL=0
MOVL C00779 V=800.0 PL=0
MOVL C00780 V=800.0 PL=0
MOVL C00781 V=800.0 PL=0
MOVL C00782 V=800.0 PL=0
MOVL C00783 V=800.0 PL=0
MOVL C00784 V=800.0 PL=0
MOVL C00785 V=800.0 PL=0
MOVL C00786 V=800.0 PL=0
MOVL C00787 V=800.0 PL=0
MOVL C00788 V=800.0 PL=0
MOVL C00789 V=800.0 PL=0
MOVL C00790 V=800.0 PL=0
MOVL C00791 V=800.0 PL=0
MOVL C00792 V=800.0 PL=0
MOVL C00793 V=800.0 PL=0
MOVL C00794 V=800.0 PL=0
MOVL C00795 V=800.0 PL=0
MOVL C00796 V=800.0 PL=0
MOVL C00797 V=800.0 PL=0
MOVL C00798 V=800.0 PL=0
MOVL C00799 V=800.0 PL=0
MOVL C00800 V=800.0 PL=0
MOVL C00801 V=800.0 PL=0
MOVL C00802 V=800.0 PL=0
MOVL C00803 V=800.0 PL=0
MOVL C00804 V=800.0 PL=0
MOVL C00805 V=800.0 PL=0
MOVL C00806 V=800.0 PL=0
MOVL C00807 V=800.0 PL=0
MOVL C00808 V=800.0 PL=0
MOVL C00809 V=800.0 PL=0
MOVL C00810 V=800.0 PL=0
MOVL C00811 V=800.0 PL=0
MOVL C00812 V=800.0 PL=0
MOVL C00813 V=800.0 PL=0
MOVL C00814 V=800.0 PL=0
MOVL C00815 V=800.0 PL=0
MOVL C00816 V=800.0 PL=0
MOVL C00817 V=800.0 PL=0
MOVL C00818 V=800.0 PL=0
MOVL C00819 V=800.0 PL=0
MOVL C00820 V=800.0 PL=0
MOVL C00821 V=800.0 PL=0
MOVL C00822 V=800.0 PL=0
MOVL C00823 V=800.0 PL=0
MOVL C00824 V=800.0 PL=0
MOVL C00825 V=800.0 PL=0
MOVL C00826 V=800.0 PL=0
MOVL C00827 V=800.0 PL=0
MOVL C00828 V=800.0 PL=0
MOVL C00829 V=800.0 PL=0
MOVL C00830 V=800.0 PL=0
MOVL C00831 V=800.0 PL=0
MOVL C00832 V=800.0 PL=0
MOVL C00833 V=800.0 PL=0
MOVL C00834 V=800.0 PL=0
MOVL C00835 V=800.0 PL=0
MOVL C00836 V=800.0 PL=0
MOVL C00837 V=800.0 PL=0
MOVL C00838 V=800.0 PL=0
MOVL C00839 V=800.0 PL=0
MOVL C00840 V=800.0 PL=0
MOVL C00841 V=800.0 PL=0
MOVL C00842 V=800.0 PL=0
MOVL C00843 V=800.0 PL=0
MOVL C00844 V=800.0 PL=0
MOVL C00845 V=800.0 PL=0
MOVL C00846 V=800.0 PL=0
MOVL C00847 V=800.0 PL=0
MOVL C00848 V=800.0 PL=0
MOVL C00849 V=800.0 PL=0
MOVL C00850 V=800.0 PL=0
MOVL C00851 V=800.0 PL=0
MOVL C00852 V=800.0 PL=0
MOVL C00853 V=800.0 PL=0
MOVL C00854 V=800.0 PL=0
MOVL C00855 V=800.0 PL=0
MOVL C00856 V=800.0 PL=0
MOVL C00857 V=800.0 PL=0
MOVL C00858 V=800.0 PL=0
MOVL C00859 V=800.0 PL=0
MOVL C00860 V=800.0 PL=0
MOVL C00861 V=800.0 PL=0
MOVL C00862 V=800.0 PL=0
MOVL C00863 V=800.0 PL=0
MOVL C00864 V=800.0 PL=0
MOVL C00865 V=800.0 PL=0
MOVL C00866 V=800.0 PL=0
MOVL C00867 V=800.0 PL=0
MOVL C00868 V=800.0 PL=0
MOVL C00869 V=800.0 PL=0
MOVL C00870 V=800.0 PL=0
MOVL C00871 V=800.0 PL=0
MOVL C00872 V=800.0 PL=0
MOVL C00873 V=800.0 PL=0
MOVL C00874 V=800.0 PL=0
MOVL C00875 V=800.0 PL=0
MOVL C00876 V=800.0 PL=0
MOVL C00877 V=800.0 PL=0
MOVL C00878 V=800.0 PL=0
MOVL C00879 V=800.0 PL=0
MOVL C00880 V=800.0 PL=0
MOVL C00881 V=800.0 PL=0
MOVL C00882 V=800.0 PL=0
MOVL C00883 V=800.0 PL=0
MOVL C00884 V=800.0 PL=0
MOVL C00885 V=800.0 PL=0
MOVL C00886 V=800.0 PL=0
MOVL C00887 V=800.0 PL=0
MOVL C00888 V=800.0 PL=0
MOVL C00889 V=800.0 PL=0
MOVL C00890 V=800.0 PL=0
MOVL C00891 V=800.0 PL=0
MOVL C00892 V=800.0 PL=0
MOVL C00893 V=800.0 PL=0
MOVL C00894 V=800.0 PL=0
MOVL C00895 V=800.0 PL=0
MOVL C00896 V=800.0 PL=0
MOVL C00897 V=800.0 PL=0
MOVL C00898 V=800.0 PL=0
MOVL C00899 V=800.0 PL=0
MOVL C00900 V=800.0 PL=0
MOVL C00901 V=800.0 PL=0
MOVL C00902 V=800.0 PL=0
MOVL C00903 V=800.0 PL=0
MOVL C00904 V=800.0 PL=0
MOVL C00905 V=800.0 PL=0
MOVL C00906 V=800.0 PL=0
MOVL C00907 V=800.0 PL=0
MOVL C00908 V=800.0 PL=0
MOVL C00909 V=800.0 PL=0
MOVL C00910 V=800.0 PL=0
MOVL C00911 V=800.0 PL=0
MOVL C00912 V=800.0 PL=0
MOVL C00913 V=800.0 PL=0
MOVL C00914 V=800.0 PL=0
MOVL C00915 V=800.0 PL=0
MOVL C00916 V=800.0 PL=0
MOVL C00917 V=800.0 PL=0
MOVL C00918 V=800.0 PL=0
MOVL C00919 V=800.0 PL=0
MOVL C00920 V=800.0 PL=0
MOVL C00921 V=800.0 PL=0
MOVL C00922 V=800.0 PL=0
MOVL C00923 V=800.0 PL=0
MOVL C00924 V=800.0 PL=0
MOVL C00925 V=800.0 PL=0
MOVL C00926 V=800.0 PL=0
MOVL C00927 V=800.0 PL=0
MOVL C00928 V=800.0 PL=0
MOVL C00929 V=800.0 PL=0
MOVL C00930 V=800.0 PL=0
MOVL C00931 V=800.0 PL=0
MOVL C00932 V=800.0 PL=0
MOVL C00933 V=800.0 PL=0
MOVL C00934 V=800.0 PL=0
MOVL C00935 V=800.0 PL=0
MOVL C00936 V=800.0 PL=0
MOVL C00937 V=800.0 PL=0
MOVL C00938 V=800.0 PL=0
MOVL C00939 V=800.0 PL=0
MOVL C00940 V=800.0 PL=0
MOVL C00941 V=800.0 PL=0
MOVL C00942 V=800.0 PL=0
MOVL C00943 V=800.0 PL=0
MOVL C00944 V=800.0 PL=0
MOVL C00945 V=800.0 PL=0
MOVL C00946 V=800.0 PL=0
MOVL C00947 V=800.0 PL=0
MOVL C00948 V=800.0 PL=0
MOVL C00949 V=800.0 PL=0
MOVL C00950 V=800.0 PL=0
MOVL C00951 V=800.0 PL=0
MOVL C00952 V=800.0 PL=0
MOVL C00953 V=800.0 PL=0
MOVL C00954 V=800.0 PL=0
MOVL C00955 V=800.0 PL=0
MOVL C00956 V=800.0 PL=0
MOVL C00957 V=800.0 PL=0
MOVL C00958 V=800.0 PL=0
MOVL C00959 V=800.0 PL=0
MOVL C00960 V=800.0 PL=0
MOVL C00961 V=800.0 PL=0
MOVL C00962 V=800.0 PL=0
MOVL C00963 V=800.0 PL=0
MOVL C00964 V=800.0 PL=0
MOVL C00965 V=800.0 PL=0
MOVL C00966 V=800.0 PL=0
MOVL C00967 V=800.0 PL=0
MOVL C00968 V=800.0 PL=0
MOVL C00969 V=800.0 PL=0
MOVL C00970 V=800.0 PL=0
MOVL C00971 V=800.0 PL=0
MOVL C00972 V=800.0 PL=0
MOVL C00973 V=800.0 PL=0
MOVL C00974 V=800.0 PL=0
MOVL C00975 V=800.0 PL=0
MOVL C00976 V=800.0 PL=0
MOVL C00977 V=800.0 PL=0
MOVL C00978 V=800.0 PL=0
MOVL C00979 V=800.0 PL=0
MOVL C00980 V=800.0 PL=0
MOVL C00981 V=800.0 PL=0
MOVL C00982 V=800.0 PL=0
MOVL C00983 V=800.0 PL=0
MOVL C00984 V=800.0 PL=0
MOVL C00985 V=800.0 PL=0
MOVL C00986 V=800.0 PL=0
MOVL C00987 V=800.0 PL=0
MOVL C00988 V=800.0 PL=0
MOVL C00989 V=800.0 PL=0
MOVL C00990 V=800.0 PL=0
MOVL C00991 V=800.0 PL=0
MOVL C00992 V=800.0 PL=0
MOVL C00993 V=800.0 PL=0
MOVL C00994 V=800.0 PL=0
MOVL C00995 V=800.0 PL=0
MOVL C00996 V=800.0 PL=0
MOVL C00997 V=800.0 PL=0
MOVL C00998 V=800.0 PL=0
MOVL C00999 V=800.0 PL=0
MOVL C01000 V=800.0 PL=0
MOVL C01001 V=800.0 PL=0
MOVL C01002 V=800.0 PL=0
MOVL C01003 V=800.0 PL=0
MOVL C01004 V=800.0 PL=0
MOVL C01005 V=800.0 PL=0
MOVL C01006 V=800.0 PL=0
MOVL C01007 V=800.0 PL=0
MOVL C01008 V=800.0 PL=0
MOVL C01009 V=800.0 PL=0
MOVL C01010 V=800.0 PL=0
MOVL C01011 V=800.0 PL=0
MOVL C01012 V=800.0 PL=0
MOVL C01013 V=800.0 PL=0
MOVL C01014 V=800.0 PL=0
MOVL C01015 V=800.0 PL=0
MOVL C01016 V=800.0 PL=0
MOVL C01017 V=800.0 PL=0
MOVL C01018 V=800.0 PL=0
MOVL C01019 V=800.0 PL=0
MOVL C01020 V=800.0 PL=0
MOVL C01021 V=800.0 PL=0
MOVL C01022 V=800.0 PL=0
MOVL C01023 V=800.0 PL=0
MOVL C01024 V=800.0 PL=0
MOVL C01025 V=800.0 PL=0
MOVL C01026 V=800.0 PL=0
MOVL C01027 V=800.0 PL=0
MOVL C01028 V=800.0 PL=0
MOVL C01029 V=800.0 PL=0
MOVL C01030 V=800.0 PL=0
MOVL C01031 V=800.0 PL=0
MOVL C01032 V=800.0 PL=0
MOVL C01033 V=800.0 PL=0
MOVL C01034 V=800.0 PL=0
MOVL C01035 V=800.0 PL=0
MOVL C01036 V=800.0 PL=0
MOVL C01037 V=800.0 PL=0
MOVL C01038 V=800.0 PL=0
MOVL C01039 V=800.0 PL=0
MOVL C01040 V=800.0 PL=0
MOVL C01041 V=800.0 PL=0
MOVL C01042 V=800.0 PL=0
MOVL C01043 V=800.0 PL=0
MOVL C01044 V=800.0 PL=0
MOVL C01045 V=800.0 PL=0
MOVL C01046 V=800.0 PL=0
MOVL C01047 V=800.0 PL=0
MOVL C01048 V=800.0 PL=0
MOVL C01049 V=800.0 PL=0
MOVL C01050 V=800.0 PL=0
MOVL C01051 V=800.0 PL=0
MOVL C01052 V=800.0 PL=0
MOVL C01053 V=800.0 PL=0
MOVL C01054 V=800.0 PL=0
MOVL C01055 V=800.0 PL=0
MOVL C01056 V=800.0 PL=0
MOVL C01057 V=800.0 PL=0
MOVL C01058 V=800.0 PL=0
MOVL C01059 V=800.0 PL=0
MOVL C01060 V=800.0 PL=0
MOVL C01061 V=800.0 PL=0
MOVL C01062 V=800.0 PL=0
MOVL C01063 V=800.0 PL=0
MOVL C01064 V=800.0 PL=0
MOVL C01065 V=800.0 PL=0
MOVL C01066 V=800.0 PL=0
MOVL C01067 V=800.0 PL=0
MOVL C01068 V=800.0 PL=0
MOVL C01069 V=800.0 PL=0
MOVL C01070 V=800.0 PL=0
MOVL C01071 V=800.0 PL=0
MOVL C01072 V=800.0 PL=0
MOVL C01073 V=800.0 PL=0
MOVL C01074 V=800.0 PL=0
MOVL C01075 V=800.0 PL=0
MOVL C01076 V=800.0 PL=0
MOVL C01077 V=800.0 PL=0
MOVL C01078 V=800.0 PL=0
MOVL C01079 V=800.0 PL=0
MOVL C01080 V=800.0 PL=0
MOVL C01081 V=800.0 PL=0
MOVL C01082 V=800.0 PL=0
MOVL C01083 V=800.0 PL=0
MOVL C01084 V=800.0 PL=0
MOVL C01085 V=800.0 PL=0
MOVL C01086 V=800.0 PL=0
MOVL C01087 V=800.0 PL=0
MOVL C01088 V=800.0 PL=0
MOVL C01089 V=800.0 PL=0
MOVL C01090 V=800.0 PL=0
MOVL C01091 V=800.0 PL=0
MOVL C01092 V=800.0 PL=0
MOVL C01093 V=800.0 PL=0
MOVL C01094 V=800.0 PL=0
MOVL C01095 V=800.0 PL=0
MOVL C01096 V=800.0 PL=0
MOVL C01097 V=800.0 PL=0
MOVL C01098 V=800.0 PL=0
MOVL C01099 V=800.0 PL=0
MOVL C01100 V=800.0 PL=0
MOVL C01101 V=800.0 PL=0
MOVL C01102 V=800.0 PL=0
MOVL C01103 V=800.0 PL=0
MOVL C01104 V=800.0 PL=0
MOVL C01105 V=800.0 PL=0
MOVL C01106 V=800.0 PL=0
MOVL C01107 V=800.0 PL=0
MOVL C01108 V=800.0 PL=0
MOVL C01109 V=800.0 PL=0
MOVL C01110 V=800.0 PL=0
MOVL C01111 V=800.0 PL=0
MOVL C01112 V=800.0 PL=0
MOVL C01113 V=800.0 PL=0
MOVL C01114 V=800.0 PL=0
MOVL C01115 V=800.0 PL=0
MOVL C01116 V=800.0 PL=0
MOVL C01117 V=800.0 PL=0
MOVL C01118 V=800.0 PL=0
MOVL C01119 V=800.0 PL=0
MOVL C01120 V=800.0 PL=0
MOVL C01121 V=800.0 PL=0
MOVL C01122 V=800.0 PL=0
MOVL C01123 V=800.0 PL=0
MOVL C01124 V=800.0 PL=0
MOVL C01125 V=800.0 PL=0
MOVL C01126 V=800.0 PL=0
MOVL C01127 V=800.0 PL=0
MOVL C01128 V=800.0 PL=0
MOVL C01129 V=800.0 PL=0
MOVL C01130 V=800.0 PL=0
MOVL C01131 V=800.0 PL=0
MOVL C01132 V=800.0 PL=0
MOVL C01133 V=800.0 PL=0
MOVL C01134 V=800.0 PL=0
MOVL C01135 V=800.0 PL=0
MOVL C01136 V=800.0 PL=0
MOVL C01137 V=800.0 PL=0
MOVL C01138 V=800.0 PL=0
MOVL C01139 V=800.0 PL=0
MOVL C01140 V=800.0 PL=0
MOVL C01141 V=800.0 PL=0
MOVL C01142 V=800.0 PL=0
MOVL C01143 V=800.0 PL=0
MOVL C01144 V=800.0 PL=0
MOVL C01145 V=800.0 PL=0
MOVL C01146 V=800.0 PL=0
MOVL C01147 V=800.0 PL=0
MOVL C01148 V=800.0 PL=0
MOVL C01149 V=800.0 PL=0
MOVL C01150 V=800.0 PL=0
MOVL C01151 V=800.0 PL=0
MOVL C01152 V=800.0 PL=0
MOVL C01153 V=800.0 PL=0
MOVL C01154 V=800.0 PL=0
MOVL C01155 V=800.0 PL=0
MOVL C01156 V=800.0 PL=0
MOVL C01157 V=800.0 PL=0
MOVL C01158 V=800.0 PL=0
MOVL C01159 V=800.0 PL=0
MOVL C01160 V=800.0 PL=0
MOVL C01161 V=800.0 PL=0
MOVL C01162 V=800.0 PL=0
MOVL C01163 V=800.0 PL=0
MOVL C01164 V=800.0 PL=0
MOVL C01165 V=800.0 PL=0
MOVL C01166 V=800.0 PL=0
MOVL C01167 V=800.0 PL=0
MOVL C01168 V=800.0 PL=0
MOVL C01169 V=800.0 PL=0
MOVL C01170 V=800.0 PL=0
MOVL C01171 V=800.0 PL=0
MOVL C01172 V=800.0 PL=0
MOVL C01173 V=800.0 PL=0
MOVL C01174 V=800.0 PL=0
MOVL C01175 V=800.0 PL=0
MOVL C01176 V=800.0 PL=0
MOVL C01177 V=800.0 PL=0
MOVL C01178 V=800.0 PL=0
MOVL C01179 V=800.0 PL=0
MOVL C01180 V=800.0 PL=0
MOVL C01181 V=800.0 PL=0
MOVL C01182 V=800.0 PL=0
MOVL C01183 V=800.0 PL=0
MOVL C01184 V=800.0 PL=0
MOVL C01185 V=800.0 PL=0
MOVL C01186 V=800.0 PL=0
MOVL C01187 V=800.0 PL=0
MOVL C01188 V=800.0 PL=0
MOVL C01189 V=800.0 PL=0
MOVL C01190 V=800.0 PL=0
MOVL C01191 V=800.0 PL=0
MOVL C01192 V=800.0 PL=0
MOVL C01193 V=800.0 PL=0
MOVL C01194 V=800.0 PL=0
MOVL C01195 V=800.0 PL=0
MOVL C01196 V=800.0 PL=0
MOVL C01197 V=800.0 PL=0
MOVL C01198 V=800.0 PL=0
MOVL C01199 V=800.0 PL=0
MOVL C01200 V=800.0 PL=0
MOVL C01201 V=800.0 PL=0
MOVL C01202 V=800.0 PL=0
MOVL C01203 V=800.0 PL=0
MOVL C01204 V=800.0 PL=0
MOVL C01205 V=800.0 PL=0
MOVL C01206 V=800.0 PL=0
MOVL C01207 V=800.0 PL=0
MOVL C01208 V=800.0 PL=0
MOVL C01209 V=800.0 PL=0
MOVL C01210 V=800.0 PL=0
MOVL C01211 V=800.0 PL=0
MOVL C01212 V=800.0 PL=0
MOVL C01213 V=800.0 PL=0
MOVL C01214 V=800.0 PL=0
MOVL C01215 V=800.0 PL=0
MOVL C01216 V=800.0 PL=0
MOVL C01217 V=800.0 PL=0
MOVL C01218 V=800.0 PL=0
MOVL C01219 V=800.0 PL=0
MOVL C01220 V=800.0 PL=0
MOVL C01221 V=800.0 PL=0
MOVL C01222 V=800.0 PL=0
MOVL C01223 V=800.0 PL=0
MOVL C01224 V=800.0 PL=0
MOVL C01225 V=800.0 PL=0
MOVL C01226 V=800.0 PL=0
MOVL C01227 V=800.0 PL=0
MOVL C01228 V=800.0 PL=0
MOVL C01229 V=800.0 PL=0
MOVL C01230 V=800.0 PL=0
MOVL C01231 V=800.0 PL=0
MOVL C01232 V=800.0 PL=0
MOVL C01233 V=800.0 PL=0
MOVL C01234 V=800.0 PL=0
MOVL C01235 V=800.0 PL=0
MOVL C01236 V=800.0 PL=0
MOVL C01237 V=800.0 PL=0
MOVL C01238 V=800.0 PL=0
MOVL C01239 V=800.0 PL=0
MOVL C01240 V=800.0 PL=0
MOVL C01241 V=800.0 PL=0
MOVL C01242 V=800.0 PL=0
MOVL C01243 V=800.0 PL=0
MOVL C01244 V=800.0 PL=0
MOVL C01245 V=800.0 PL=0
MOVL C01246 V=800.0 PL=0
MOVL C01247 V=800.0 PL=0
MOVL C01248 V=800.0 PL=0
MOVL C01249 V=800.0 PL=0
MOVL C01250 V=800.0 PL=0
MOVL C01251 V=800.0 PL=0
MOVL C01252 V=800.0 PL=0
MOVL C01253 V=800.0 PL=0
MOVL C01254 V=800.0 PL=0
MOVL C01255 V=800.0 PL=0
MOVL C01256 V=800.0 PL=0
MOVL C01257 V=800.0 PL=0
MOVL C01258 V=800.0 PL=0
MOVL C01259 V=800.0 PL=0
MOVL C01260 V=800.0 PL=0
MOVL C01261 V=800.0 PL=0
MOVL C01262 V=800.0 PL=0
MOVL C01263 V=800.0 PL=0
MOVL C01264 V=800.0 PL=0
MOVL C01265 V=800.0 PL=0
MOVL C01266 V=800.0 PL=0
MOVL C01267 V=800.0 PL=0
MOVL C01268 V=800.0 PL=0
MOVL C01269 V=800.0 PL=0
MOVL C01270 V=800.0 PL=0
MOVL C01271 V=800.0 PL=0
MOVL C01272 V=800.0 PL=0
MOVL C01273 V=800.0 PL=0
MOVL C01274 V=800.0 PL=0
MOVL C01275 V=800.0 PL=0
MOVL C01276 V=800.0 PL=0
MOVL C01277 V=800.0 PL=0
MOVL C01278 V=800.0 PL=0
MOVL C01279 V=800.0 PL=0
MOVL C01280 V=800.0 PL=0
MOVL C01281 V=800.0 PL=0
MOVL C01282 V=800.0 PL=0
MOVL C01283 V=800.0 PL=0
MOVL C01284 V=800.0 PL=0
MOVL C01285 V=800.0 PL=0
MOVL C01286 V=800.0 PL=0
MOVL C01287 V=800.0 PL=0
MOVL C01288 V=800.0 PL=0
MOVL C01289 V=800.0 PL=0
MOVL C01290 V=800.0 PL=0
MOVL C01291 V=800.0 PL=0
MOVL C01292 V=800.0 PL=0
MOVL C01293 V=800.0 PL=0
MOVL C01294 V=800.0 PL=0
MOVL C01295 V=800.0 PL=0
MOVL C01296 V=800.0 PL=0
MOVL C01297 V=800.0 PL=0
MOVL C01298 V=800.0 PL=0
MOVL C01299 V=800.0 PL=0
MOVL C01300 V=800.0 PL=0
MOVL C01301 V=800.0 PL=0
MOVL C01302 V=800.0 PL=0
MOVL C01303 V=800.0 PL=0
MOVL C01304 V=800.0 PL=0
MOVL C01305 V=800.0 PL=0
MOVL C01306 V=800.0 PL=0
MOVL C01307 V=800.0 PL=0
MOVL C01308 V=800.0 PL=0
MOVL C01309 V=800.0 PL=0
MOVL C01310 V=800.0 PL=0
MOVL C01311 V=800.0 PL=0
MOVL C01312 V=800.0 PL=0
MOVL C01313 V=800.0 PL=0
MOVL C01314 V=800.0 PL=0
MOVL C01315 V=800.0 PL=0
MOVL C01316 V=800.0 PL=0
MOVL C01317 V=800.0 PL=0
MOVL C01318 V=800.0 PL=0
MOVL C01319 V=800.0 PL=0
MOVL C01320 V=800.0 PL=0
MOVL C01321 V=800.0 PL=0
MOVL C01322 V=800.0 PL=0
MOVL C01323 V=800.0 PL=0
MOVL C01324 V=800.0 PL=0
MOVL C01325 V=800.0 PL=0
MOVL C01326 V=800.0 PL=0
MOVL C01327 V=800.0 PL=0
MOVL C01328 V=800.0 PL=0
MOVL C01329 V=800.0 PL=0
MOVL C01330 V=800.0 PL=0
MOVL C01331 V=800.0 PL=0
MOVL C01332 V=800.0 PL=0
MOVL C01333 V=800.0 PL=0
MOVL C01334 V=800.0 PL=0
MOVL C01335 V=800.0 PL=0
MOVL C01336 V=800.0 PL=0
MOVL C01337 V=800.0 PL=0
MOVL C01338 V=800.0 PL=0
MOVL C01339 V=800.0 PL=0
MOVL C01340 V=800.0 PL=0
MOVL C01341 V=800.0 PL=0
MOVL C01342 V=800.0 PL=0
MOVL C01343 V=800.0 PL=0
MOVL C01344 V=800.0 PL=0
MOVL C01345 V=800.0 PL=0
MOVL C01346 V=800.0 PL=0
MOVL C01347 V=800.0 PL=0
MOVL C01348 V=800.0 PL=0
MOVL C01349 V=800.0 PL=0
MOVL C01350 V=800.0 PL=0
MOVL C01351 V=800.0 PL=0
MOVL C01352 V=800.0 PL=0
MOVL C01353 V=800.0 PL=0
MOVL C01354 V=800.0 PL=0
MOVL C01355 V=800.0 PL=0
MOVL C01356 V=800.0 PL=0
MOVL C01357 V=800.0 PL=0
MOVL C01358 V=800.0 PL=0
MOVL C01359 V=800.0 PL=0
MOVL C01360 V=800.0 PL=0
MOVL C01361 V=800.0 PL=0
MOVL C01362 V=800.0 PL=0
MOVL C01363 V=800.0 PL=0
MOVL C01364 V=800.0 PL=0
MOVL C01365 V=800.0 PL=0
MOVL C01366 V=800.0 PL=0
MOVL C01367 V=800.0 PL=0
MOVL C01368 V=800.0 PL=0
MOVL C01369 V=800.0 PL=0
MOVL C01370 V=800.0 PL=0
MOVL C01371 V=800.0 PL=0
MOVL C01372 V=800.0 PL=0
MOVL C01373 V=800.0 PL=0
MOVL C01374 V=800.0 PL=0
MOVL C01375 V=800.0 PL=0
MOVL C01376 V=800.0 PL=0
MOVL C01377 V=800.0 PL=0
MOVL C01378 V=800.0 PL=0
MOVL C01379 V=800.0 PL=0
MOVL C01380 V=800.0 PL=0
MOVL C01381 V=800.0 PL=0
MOVL C01382 V=800.0 PL=0
MOVL C01383 V=800.0 PL=0
MOVL C01384 V=800.0 PL=0
MOVL C01385 V=800.0 PL=0
MOVL C01386 V=800.0 PL=0
MOVL C01387 V=800.0 PL=0
MOVL C01388 V=800.0 PL=0
MOVL C01389 V=800.0 PL=0
MOVL C01390 V=800.0 PL=0
MOVL C01391 V=800.0 PL=0
MOVL C01392 V=800.0 PL=0
MOVL C01393 V=800.0 PL=0
MOVL C01394 V=800.0 PL=0
MOVL C01395 V=800.0 PL=0
MOVL C01396 V=800.0 PL=0
MOVL C01397 V=800.0 PL=0
MOVL C01398 V=800.0 PL=0
MOVL C01399 V=800.0 PL=0
MOVL C01400 V=800.0 PL=0
MOVL C01401 V=800.0 PL=0
MOVL C01402 V=800.0 PL=0
MOVL C01403 V=800.0 PL=0
MOVL C01404 V=800.0 PL=0
MOVL C01405 V=800.0 PL=0
MOVL C01406 V=800.0 PL=0
MOVL C01407 V=800.0 PL=0
MOVL C01408 V=800.0 PL=0
MOVL C01409 V=800.0 PL=0
MOVL C01410 V=800.0 PL=0
MOVL C01411 V=800.0 PL=0
MOVL C01412 V=800.0 PL=0
MOVL C01413 V=800.0 PL=0
MOVL C01414 V=800.0 PL=0
MOVL C01415 V=800.0 PL=0
MOVL C01416 V=800.0 PL=0
MOVL C01417 V=800.0 PL=0
MOVL C01418 V=800.0 PL=0
MOVL C01419 V=800.0 PL=0
MOVL C01420 V=800.0 PL=0
MOVL C01421 V=800.0 PL=0
MOVL C01422 V=800.0 PL=0
MOVL C01423 V=800.0 PL=0
MOVL C01424 V=800.0 PL=0
MOVL C01425 V=800.0 PL=0
MOVL C01426 V=800.0 PL=0
MOVL C01427 V=800.0 PL=0
MOVL C01428 V=800.0 PL=0
MOVL C01429 V=800.0 PL=0
MOVL C01430 V=800.0 PL=0
MOVL C01431 V=800.0 PL=0
MOVL C01432 V=800.0 PL=0
MOVL C01433 V=800.0 PL=0
MOVL C01434 V=800.0 PL=0
MOVL C01435 V=800.0 PL=0
MOVL C01436 V=800.0 PL=0
MOVL C01437 V=800.0 PL=0
MOVL C01438 V=800.0 PL=0
MOVL C01439 V=800.0 PL=0
MOVL C01440 V=800.0 PL=0
MOVL C01441 V=800.0 PL=0
MOVL C01442 V=800.0 PL=0
MOVL C01443 V=800.0 PL=0
MOVL C01444 V=800.0 PL=0
MOVL C01445 V=800.0 PL=0
MOVL C01446 V=800.0 PL=0
MOVL C01447 V=800.0 PL=0
MOVL C01448 V=800.0 PL=0
MOVL C01449 V=800.0 PL=0
MOVL C01450 V=800.0 PL=0
MOVL C01451 V=800.0 PL=0
MOVL C01452 V=800.0 PL=0
MOVL C01453 V=800.0 PL=0
MOVL C01454 V=800.0 PL=0
MOVL C01455 V=800.0 PL=0
MOVL C01456 V=800.0 PL=0
MOVL C01457 V=800.0 PL=0
MOVL C01458 V=800.0 PL=0
MOVL C01459 V=800.0 PL=0
MOVL C01460 V=800.0 PL=0
MOVL C01461 V=800.0 PL=0
MOVL C01462 V=800.0 PL=0
MOVL C01463 V=800.0 PL=0
MOVL C01464 V=800.0 PL=0
MOVL C01465 V=800.0 PL=0
MOVL C01466 V=800.0 PL=0
MOVL C01467 V=800.0 PL=0
MOVL C01468 V=800.0 PL=0
MOVL C01469 V=800.0 PL=0
MOVL C01470 V=800.0 PL=0
MOVL C01471 V=800.0 PL=0
MOVL C01472 V=800.0 PL=0
MOVL C01473 V=800.0 PL=0
MOVL C01474 V=800.0 PL=0
MOVL C01475 V=800.0 PL=0
MOVL C01476 V=800.0 PL=0
MOVL C01477 V=800.0 PL=0
MOVL C01478 V=800.0 PL=0
MOVL C01479 V=800.0 PL=0
MOVL C01480 V=800.0 PL=0
MOVL C01481 V=800.0 PL=0
MOVL C01482 V=800.0 PL=0
MOVL C01483 V=800.0 PL=0
MOVL C01484 V=800.0 PL=0
MOVL C01485 V=800.0 PL=0
MOVL C01486 V=800.0 PL=0
MOVL C01487 V=800.0 PL=0
MOVL C01488 V=800.0 PL=0
MOVL C01489 V=800.0 PL=0
MOVL C01490 V=800.0 PL=0
MOVL C01491 V=800.0 PL=0
MOVL C01492 V=800.0 PL=0
MOVL C01493 V=800.0 PL=0
MOVL C01494 V=800.0 PL=0
MOVL C01495 V=800.0 PL=0
MOVL C01496 V=800.0 PL=0
MOVL C01497 V=800.0 PL=0
MOVL C01498 V=800.0 PL=0
MOVL C01499 V=800.0 PL=0
MOVL C01500 V=800.0 PL=0
MOVL C01501 V=800.0 PL=0
MOVL C01502 V=800.0 PL=0
MOVL C01503 V=800.0 PL=0
MOVL C01504 V=800.0 PL=0
MOVL C01505 V=800.0 PL=0
MOVL C01506 V=800.0 PL=0
MOVL C01507 V=800.0 PL=0
MOVL C01508 V=800.0 PL=0
MOVL C01509 V=800.0 PL=0
MOVL C01510 V=800.0 PL=0
MOVL C01511 V=800.0 PL=0
MOVL C01512 V=800.0 PL=0
MOVL C01513 V=800.0 PL=0
MOVL C01514 V=800.0 PL=0
MOVL C01515 V=800.0 PL=0
MOVL C01516 V=800.0 PL=0
MOVL C01517 V=800.0 PL=0
MOVL C01518 V=800.0 PL=0
MOVL C01519 V=800.0 PL=0
MOVL C01520 V=800.0 PL=0
MOVL C01521 V=800.0 PL=0
MOVL C01522 V=800.0 PL=0
MOVL C01523 V=800.0 PL=0
MOVL C01524 V=800.0 PL=0
MOVL C01525 V=800.0 PL=0
MOVL C01526 V=800.0 PL=0
MOVL C01527 V=800.0 PL=0
MOVL C01528 V=800.0 PL=0
MOVL C01529 V=800.0 PL=0
MOVL C01530 V=800.0 PL=0
MOVL C01531 V=800.0 PL=0
MOVL C01532 V=800.0 PL=0
MOVL C01533 V=800.0 PL=0
MOVL C01534 V=800.0 PL=0
MOVL C01535 V=800.0 PL=0
MOVL C01536 V=800.0 PL=0
MOVL C01537 V=800.0 PL=0
MOVL C01538 V=800.0 PL=0
MOVL C01539 V=800.0 PL=0
MOVL C01540 V=800.0 PL=0
MOVL C01541 V=800.0 PL=0
MOVL C01542 V=800.0 PL=0
MOVL C01543 V=800.0 PL=0
MOVL C01544 V=800.0 PL=0
MOVL C01545 V=800.0 PL=0
MOVL C01546 V=800.0 PL=0
MOVL C01547 V=800.0 PL=0
MOVL C01548 V=800.0 PL=0
MOVL C01549 V=800.0 PL=0
MOVL C01550 V=800.0 PL=0
MOVL C01551 V=800.0 PL=0
MOVL C01552 V=800.0 PL=0
MOVL C01553 V=800.0 PL=0
MOVL C01554 V=800.0 PL=0
MOVL C01555 V=800.0 PL=0
MOVL C01556 V=800.0 PL=0
MOVL C01557 V=800.0 PL=0
MOVL C01558 V=800.0 PL=0
MOVL C01559 V=800.0 PL=0
MOVL C01560 V=800.0 PL=0
MOVL C01561 V=800.0 PL=0
MOVL C01562 V=800.0 PL=0
MOVL C01563 V=800.0 PL=0
MOVL C01564 V=800.0 PL=0
MOVL C01565 V=800.0 PL=0
MOVL C01566 V=800.0 PL=0
MOVL C01567 V=800.0 PL=0
MOVL C01568 V=800.0 PL=0
MOVL C01569 V=800.0 PL=0
MOVL C01570 V=800.0 PL=0
MOVL C01571 V=800.0 PL=0
MOVL C01572 V=800.0 PL=0
MOVL C01573 V=800.0 PL=0
MOVL C01574 V=800.0 PL=0
MOVL C01575 V=800.0 PL=0
MOVL C01576 V=800.0 PL=0
MOVL C01577 V=800.0 PL=0
MOVL C01578 V=800.0 PL=0
MOVL C01579 V=800.0 PL=0
MOVL C01580 V=800.0 PL=0
MOVL C01581 V=800.0 PL=0
MOVL C01582 V=800.0 PL=0
MOVL C01583 V=800.0 PL=0
MOVL C01584 V=800.0 PL=0
MOVL C01585 V=800.0 PL=0
MOVL C01586 V=800.0 PL=0
MOVL C01587 V=800.0 PL=0
MOVL C01588 V=800.0 PL=0
MOVL C01589 V=800.0 PL=0
MOVL C01590 V=800.0 PL=0
MOVL C01591 V=800.0 PL=0
MOVL C01592 V=800.0 PL=0
MOVL C01593 V=800.0 PL=0
MOVL C01594 V=800.0 PL=0
MOVL C01595 V=800.0 PL=0
MOVL C01596 V=800.0 PL=0
MOVL C01597 V=800.0 PL=0
MOVL C01598 V=800.0 PL=0
MOVL C01599 V=800.0 PL=0
MOVL C01600 V=800.0 PL=0
MOVL C01601 V=800.0 PL=0
MOVL C01602 V=800.0 PL=0
MOVL C01603 V=800.0 PL=0
MOVL C01604 V=800.0 PL=0
MOVL C01605 V=800.0 PL=0
MOVL C01606 V=800.0 PL=0
MOVL C01607 V=800.0 PL=0
MOVL C01608 V=800.0 PL=0
MOVL C01609 V=800.0 PL=0
MOVL C01610 V=800.0 PL=0
MOVL C01611 V=800.0 PL=0
MOVL C01612 V=800.0 PL=0
MOVL C01613 V=800.0 PL=0
MOVL C01614 V=800.0 PL=0
MOVL C01615 V=800.0 PL=0
MOVL C01616 V=800.0 PL=0
MOVL C01617 V=800.0 PL=0
MOVL C01618 V=800.0 PL=0
MOVL C01619 V=800.0 PL=0
MOVL C01620 V=800.0 PL=0
MOVL C01621 V=800.0 PL=0
MOVL C01622 V=800.0 PL=0
MOVL C01623 V=800.0 PL=0
MOVL C01624 V=800.0 PL=0
MOVL C01625 V=800.0 PL=0
MOVL C01626 V=800.0 PL=0
MOVL C01627 V=800.0 PL=0
MOVL C01628 V=800.0 PL=0
MOVL C01629 V=800.0 PL=0
MOVL C01630 V=800.0 PL=0
MOVL C01631 V=800.0 PL=0
MOVL C01632 V=800.0 PL=0
MOVL C01633 V=800.0 PL=0
MOVL C01634 V=800.0 PL=0
MOVL C01635 V=800.0 PL=0
MOVL C01636 V=800.0 PL=0
MOVL C01637 V=800.0 PL=0
MOVL C01638 V=800.0 PL=0
MOVL C01639 V=800.0 PL=0
MOVL C01640 V=800.0 PL=0
MOVL C01641 V=800.0 PL=0
MOVL C01642 V=800.0 PL=0
MOVL C01643 V=800.0 PL=0
MOVL C01644 V=800.0 PL=0
MOVL C01645 V=800.0 PL=0
MOVL C01646 V=800.0 PL=0
MOVL C01647 V=800.0 PL=0
MOVL C01648 V=800.0 PL=0
MOVL C01649 V=800.0 PL=0
MOVL C01650 V=800.0 PL=0
MOVL C01651 V=800.0 PL=0
MOVL C01652 V=800.0 PL=0
MOVL C01653 V=800.0 PL=0
MOVL C01654 V=800.0 PL=0
MOVL C01655 V=800.0 PL=0
MOVL C01656 V=800.0 PL=0
MOVL C01657 V=800.0 PL=0
MOVL C01658 V=800.0 PL=0
MOVL C01659 V=800.0 PL=0
MOVL C01660 V=800.0 PL=0
MOVL C01661 V=800.0 PL=0
MOVL C01662 V=800.0 PL=0
MOVL C01663 V=800.0 PL=0
MOVL C01664 V=800.0 PL=0
MOVL C01665 V=800.0 PL=0
MOVL C01666 V=800.0 PL=0
MOVL C01667 V=800.0 PL=0
MOVL C01668 V=800.0 PL=0
MOVL C01669 V=800.0 PL=0
MOVL C01670 V=800.0 PL=0
MOVL C01671 V=800.0 PL=0
MOVL C01672 V=800.0 PL=0
MOVL C01673 V=800.0 PL=0
MOVL C01674 V=800.0 PL=0
MOVL C01675 V=800.0 PL=0
MOVL C01676 V=800.0 PL=0
MOVL C01677 V=800.0 PL=0
MOVL C01678 V=800.0 PL=0
MOVL C01679 V=800.0 PL=0
MOVL C01680 V=800.0 PL=0
MOVL C01681 V=800.0 PL=0
MOVL C01682 V=800.0 PL=0
MOVL C01683 V=800.0 PL=0
MOVL C01684 V=800.0 PL=0
MOVL C01685 V=800.0 PL=0
MOVL C01686 V=800.0 PL=0
MOVL C01687 V=800.0 PL=0
MOVL C01688 V=800.0 PL=0
MOVL C01689 V=800.0 PL=0
MOVL C01690 V=800.0 PL=0
MOVL C01691 V=800.0 PL=0
MOVL C01692 V=800.0 PL=0
MOVL C01693 V=800.0 PL=0
MOVL C01694 V=800.0 PL=0
MOVL C01695 V=800.0 PL=0
MOVL C01696 V=800.0 PL=0
MOVL C01697 V=800.0 PL=0
MOVL C01698 V=800.0 PL=0
MOVL C01699 V=800.0 PL=0
MOVL C01700 V=800.0 PL=0
MOVL C01701 V=800.0 PL=0
MOVL C01702 V=800.0 PL=0
MOVL C01703 V=800.0 PL=0
MOVL C01704 V=800.0 PL=0
MOVL C01705 V=800.0 PL=0
MOVL C01706 V=800.0 PL=0
MOVL C01707 V=800.0 PL=0
MOVL C01708 V=800.0 PL=0
MOVL C01709 V=800.0 PL=0
MOVL C01710 V=800.0 PL=0
MOVL C01711 V=800.0 PL=0
MOVL C01712 V=800.0 PL=0
MOVL C01713 V=800.0 PL=0
MOVL C01714 V=800.0 PL=0
MOVL C01715 V=800.0 PL=0
MOVL C01716 V=800.0 PL=0
MOVL C01717 V=800.0 PL=0
MOVL C01718 V=800.0 PL=0
MOVL C01719 V=800.0 PL=0
MOVL C01720 V=800.0 PL=0
MOVL C01721 V=800.0 PL=0
MOVL C01722 V=800.0 PL=0
MOVL C01723 V=800.0 PL=0
MOVL C01724 V=800.0 PL=0
MOVL C01725 V=800.0 PL=0
MOVL C01726 V=800.0 PL=0
MOVL C01727 V=800.0 PL=0
MOVL C01728 V=800.0 PL=0
MOVL C01729 V=800.0 PL=0
MOVL C01730 V=800.0 PL=0
MOVL C01731 V=800.0 PL=0
MOVL C01732 V=800.0 PL=0
MOVL C01733 V=800.0 PL=0
MOVL C01734 V=800.0 PL=0
MOVL C01735 V=800.0 PL=0
MOVL C01736 V=800.0 PL=0
MOVL C01737 V=800.0 PL=0
MOVL C01738 V=800.0 PL=0
MOVL C01739 V=800.0 PL=0
MOVL C01740 V=800.0 PL=0
MOVL C01741 V=800.0 PL=0
MOVL C01742 V=800.0 PL=0
MOVL C01743 V=800.0 PL=0
MOVL C01744 V=800.0 PL=0
MOVL C01745 V=800.0 PL=0
MOVL C01746 V=800.0 PL=0
MOVL C01747 V=800.0 PL=0
MOVL C01748 V=800.0 PL=0
MOVL C01749 V=800.0 PL=0
MOVL C01750 V=800.0 PL=0
MOVL C01751 V=800.0 PL=0
MOVL C01752 V=800.0 PL=0
MOVL C01753 V=800.0 PL=0
MOVL C01754 V=800.0 PL=0
MOVL C01755 V=800.0 PL=0
MOVL C01756 V=800.0 PL=0
MOVL C01757 V=800.0 PL=0
MOVL C01758 V=800.0 PL=0
MOVL C01759 V=800.0 PL=0
MOVL C01760 V=800.0 PL=0
MOVL C01761 V=800.0 PL=0
MOVL C01762 V=800.0 PL=0
MOVL C01763 V=800.0 PL=0
MOVL C01764 V=800.0 PL=0
MOVL C01765 V=800.0 PL=0
MOVL C01766 V=800.0 PL=0
MOVL C01767 V=800.0 PL=0
MOVL C01768 V=800.0 PL=0
MOVL C01769 V=800.0 PL=0
MOVL C01770 V=800.0 PL=0
MOVL C01771 V=800.0 PL=0
MOVL C01772 V=800.0 PL=0
MOVL C01773 V=800.0 PL=0
MOVL C01774 V=800.0 PL=0
MOVL C01775 V=800.0 PL=0
MOVL C01776 V=800.0 PL=0
MOVL C01777 V=800.0 PL=0
MOVL C01778 V=800.0 PL=0
MOVL C01779 V=800.0 PL=0
MOVL C01780 V=800.0 PL=0
MOVL C01781 V=800.0 PL=0
MOVL C01782 V=800.0 PL=0
MOVL C01783 V=800.0 PL=0
MOVL C01784 V=800.0 PL=0
MOVL C01785 V=800.0 PL=0
MOVL C01786 V=800.0 PL=0
MOVL C01787 V=800.0 PL=0
MOVL C01788 V=800.0 PL=0
MOVL C01789 V=800.0 PL=0
MOVL C01790 V=800.0 PL=0
MOVL C01791 V=800.0 PL=0
MOVL C01792 V=800.0 PL=0
MOVL C01793 V=800.0 PL=0
MOVL C01794 V=800.0 PL=0
MOVL C01795 V=800.0 PL=0
MOVL C01796 V=800.0 PL=0
MOVL C01797 V=800.0 PL=0
MOVL C01798 V=800.0 PL=0
MOVL C01799 V=800.0 PL=0
MOVL C01800 V=800.0 PL=0
MOVL C01801 V=800.0 PL=0
MOVL C01802 V=800.0 PL=0
MOVL C01803 V=800.0 PL=0
MOVL C01804 V=800.0 PL=0
MOVL C01805 V=800.0 PL=0
MOVL C01806 V=800.0 PL=0
MOVL C01807 V=800.0 PL=0
MOVL C01808 V=800.0 PL=0
MOVL C01809 V=800.0 PL=0
MOVL C01810 V=800.0 PL=0
MOVL C01811 V=800.0 PL=0
MOVL C01812 V=800.0 PL=0
MOVL C01813 V=800.0 PL=0
MOVL C01814 V=800.0 PL=0
MOVL C01815 V=800.0 PL=0
MOVL C01816 V=800.0 PL=0
MOVL C01817 V=800.0 PL=0
MOVL C01818 V=800.0 PL=0
MOVL C01819 V=800.0 PL=0
MOVL C01820 V=800.0 PL=0
MOVL C01821 V=800.0 PL=0
MOVL C01822 V=800.0 PL=0
MOVL C01823 V=800.0 PL=0
MOVL C01824 V=800.0 PL=0
MOVL C01825 V=800.0 PL=0
MOVL C01826 V=800.0 PL=0
MOVL C01827 V=800.0 PL=0
MOVL C01828 V=800.0 PL=0
MOVL C01829 V=800.0 PL=0
MOVL C01830 V=800.0 PL=0
MOVL C01831 V=800.0 PL=0
MOVL C01832 V=800.0 PL=0
MOVL C01833 V=800.0 PL=0
MOVL C01834 V=800.0 PL=0
MOVL C01835 V=800.0 PL=0
MOVL C01836 V=800.0 PL=0
MOVL C01837 V=800.0 PL=0
MOVL C01838 V=800.0 PL=0
MOVL C01839 V=800.0 PL=0
MOVL C01840 V=800.0 PL=0
MOVL C01841 V=800.0 PL=0
MOVL C01842 V=800.0 PL=0
MOVL C01843 V=800.0 PL=0
MOVL C01844 V=800.0 PL=0
MOVL C01845 V=800.0 PL=0
MOVL C01846 V=800.0 PL=0
MOVL C01847 V=800.0 PL=0
MOVL C01848 V=800.0 PL=0
MOVL C01849 V=800.0 PL=0
MOVL C01850 V=800.0 PL=0
MOVL C01851 V=800.0 PL=0
MOVL C01852 V=800.0 PL=0
MOVL C01853 V=800.0 PL=0
MOVL C01854 V=800.0 PL=0
MOVL C01855 V=800.0 PL=0
MOVL C01856 V=800.0 PL=0
MOVL C01857 V=800.0 PL=0
MOVL C01858 V=800.0 PL=0
MOVL C01859 V=800.0 PL=0
MOVL C01860 V=800.0 PL=0
MOVL C01861 V=800.0 PL=0
MOVL C01862 V=800.0 PL=0
MOVL C01863 V=800.0 PL=0
MOVL C01864 V=800.0 PL=0
MOVL C01865 V=800.0 PL=0
MOVL C01866 V=800.0 PL=0
MOVL C01867 V=800.0 PL=0
MOVL C01868 V=800.0 PL=0
MOVL C01869 V=800.0 PL=0
MOVL C01870 V=800.0 PL=0
MOVL C01871 V=800.0 PL=0
MOVL C01872 V=800.0 PL=0
MOVL C01873 V=800.0 PL=0
MOVL C01874 V=800.0 PL=0
MOVL C01875 V=800.0 PL=0
MOVL C01876 V=800.0 PL=0
MOVL C01877 V=800.0 PL=0
MOVL C01878 V=800.0 PL=0
MOVL C01879 V=800.0 PL=0
MOVL C01880 V=800.0 PL=0
MOVL C01881 V=800.0 PL=0
MOVL C01882 V=800.0 PL=0
MOVL C01883 V=800.0 PL=0
MOVL C01884 V=800.0 PL=0
MOVL C01885 V=800.0 PL=0
MOVL C01886 V=800.0 PL=0
MOVL C01887 V=800.0 PL=0
MOVL C01888 V=800.0 PL=0
MOVL C01889 V=800.0 PL=0
MOVL C01890 V=800.0 PL=0
MOVL C01891 V=800.0 PL=0
MOVL C01892 V=800.0 PL=0
MOVL C01893 V=800.0 PL=0
MOVL C01894 V=800.0 PL=0
MOVL C01895 V=800.0 PL=0
MOVL C01896 V=800.0 PL=0
MOVL C01897 V=800.0 PL=0
MOVL C01898 V=800.0 PL=0
MOVL C01899 V=800.0 PL=0
MOVL C01900 V=800.0 PL=0
MOVL C01901 V=800.0 PL=0
MOVL C01902 V=800.0 PL=0
MOVL C01903 V=800.0 PL=0
MOVL C01904 V=800.0 PL=0
MOVL C01905 V=800.0 PL=0
MOVL C01906 V=800.0 PL=0
MOVL C01907 V=800.0 PL=0
MOVL C01908 V=800.0 PL=0
MOVL C01909 V=800.0 PL=0
MOVL C01910 V=800.0 PL=0
MOVL C01911 V=800.0 PL=0
MOVL C01912 V=800.0 PL=0
MOVL C01913 V=800.0 PL=0
MOVL C01914 V=800.0 PL=0
MOVL C01915 V=800.0 PL=0
MOVL C01916 V=800.0 PL=0
MOVL C01917 V=800.0 PL=0
MOVL C01918 V=800.0 PL=0
MOVL C01919 V=800.0 PL=0
MOVL C01920 V=800.0 PL=0
MOVL C01921 V=800.0 PL=0
MOVL C01922 V=800.0 PL=0
MOVL C01923 V=800.0 PL=0
MOVL C01924 V=800.0 PL=0
MOVL C01925 V=800.0 PL=0
MOVL C01926 V=800.0 PL=0
MOVL C01927 V=800.0 PL=0
MOVL C01928 V=800.0 PL=0
MOVL C01929 V=800.0 PL=0
MOVL C01930 V=800.0 PL=0
MOVL C01931 V=800.0 PL=0
MOVL C01932 V=800.0 PL=0
MOVL C01933 V=800.0 PL=0
MOVL C01934 V=800.0 PL=0
MOVL C01935 V=800.0 PL=0
MOVL C01936 V=800.0 PL=0
MOVL C01937 V=800.0 PL=0
MOVL C01938 V=800.0 PL=0
MOVL C01939 V=800.0 PL=0
MOVL C01940 V=800.0 PL=0
MOVL C01941 V=800.0 PL=0
MOVL C01942 V=800.0 PL=0
MOVL C01943 V=800.0 PL=0
MOVL C01944 V=800.0 PL=0
MOVL C01945 V=800.0 PL=0
MOVL C01946 V=800.0 PL=0
MOVL C01947 V=800.0 PL=0
MOVL C01948 V=800.0 PL=0
MOVL C01949 V=800.0 PL=0
MOVL C01950 V=800.0 PL=0
MOVL C01951 V=800.0 PL=0
MOVL C01952 V=800.0 PL=0
MOVL C01953 V=800.0 PL=0
MOVL C01954 V=800.0 PL=0
MOVL C01955 V=800.0 PL=0
MOVL C01956 V=800.0 PL=0
MOVL C01957 V=800.0 PL=0
MOVL C01958 V=800.0 PL=0
MOVL C01959 V=800.0 PL=0
MOVL C01960 V=800.0 PL=0
MOVL C01961 V=800.0 PL=0
MOVL C01962 V=800.0 PL=0
MOVL C01963 V=800.0 PL=0
MOVL C01964 V=800.0 PL=0
MOVL C01965 V=800.0 PL=0
MOVL C01966 V=800.0 PL=0
MOVL C01967 V=800.0 PL=0
MOVL C01968 V=800.0 PL=0
MOVL C01969 V=800.0 PL=0
MOVL C01970 V=800.0 PL=0
MOVL C01971 V=800.0 PL=0
MOVL C01972 V=800.0 PL=0
MOVL C01973 V=800.0 PL=0
MOVL C01974 V=800.0 PL=0
MOVL C01975 V=800.0 PL=0
MOVL C01976 V=800.0 PL=0
MOVL C01977 V=800.0 PL=0
MOVL C01978 V=800.0 PL=0
MOVL C01979 V=800.0 PL=0
MOVL C01980 V=800.0 PL=0
MOVL C01981 V=800.0 PL=0
MOVL C01982 V=800.0 PL=0
MOVL C01983 V=800.0 PL=0
MOVL C01984 V=800.0 PL=0
MOVL C01985 V=800.0 PL=0
MOVL C01986 V=800.0 PL=0
MOVL C01987 V=800.0 PL=0
MOVL C01988 V=800.0 PL=0
MOVL C01989 V=800.0 PL=0
MOVL C01990 V=800.0 PL=0
MOVL C01991 V=800.0 PL=0
MOVL C01992 V=800.0 PL=0
MOVL C01993 V=800.0 PL=0
MOVL C01994 V=800.0 PL=0
MOVL C01995 V=800.0 PL=0
